	REGION ReadData()
	    //************************************************************************************************ 
	    //从接口读取数据/Read data from interface
	    //************************************************************************************************ 
	    //命令状态/Command Status bits
	    #aRetvalRead[1] := DPRD_DAT(LADDR := "DB_KeyenceCheckerIV3".aDev[#I_nID].Para.nInAdr1, RECORD => #aInput_Byte1);
	    //设备结果/Device Results bits
	    #aRetvalRead[2] := DPRD_DAT(LADDR := "DB_KeyenceCheckerIV3".aDev[#I_nID].Para.nInAdr2, RECORD => #aInput_Byte2);
	    //设备状态/Device status words
	    #aRetvalRead[3] := DPRD_DAT(LADDR := "DB_KeyenceCheckerIV3".aDev[#I_nID].Para.nInAdr3, RECORD => #aInput_Byte3);
	    //设备统计/Device statistics
	    #aRetvalRead[4] := DPRD_DAT(LADDR := "DB_KeyenceCheckerIV3".aDev[#I_nID].Para.nInAdr4, RECORD => #aInput_Byte4);
	    //位置修正结果/Position adjust result
	    #aRetvalRead[5] := DPRD_DAT(LADDR := "DB_KeyenceCheckerIV3".aDev[#I_nID].Para.nInAdr5, RECORD => #aInput_Byte5);
	    //工具1处理结果/Tool1 result
	    #aRetvalRead[6] := DPRD_DAT(LADDR := "DB_KeyenceCheckerIV3".aDev[#I_nID].Para.nInAdr6, RECORD => #aInput_Byte6[0]);
	    //工具2处理结果/Tool2 result
	    #aRetvalRead[7] := DPRD_DAT(LADDR := "DB_KeyenceCheckerIV3".aDev[#I_nID].Para.nInAdr7, RECORD => #aInput_Byte6[1]);
	    //工具3处理结果/Tool3 result
	    #aRetvalRead[8] := DPRD_DAT(LADDR := "DB_KeyenceCheckerIV3".aDev[#I_nID].Para.nInAdr8, RECORD => #aInput_Byte6[2]);
	    //工具4处理结果/Tool4 result
	    #aRetvalRead[9] := DPRD_DAT(LADDR := "DB_KeyenceCheckerIV3".aDev[#I_nID].Para.nInAdr9, RECORD => #aInput_Byte6[3]);
	    //工具5处理结果/Tool5 result
	    #aRetvalRead[10] := DPRD_DAT(LADDR := "DB_KeyenceCheckerIV3".aDev[#I_nID].Para.nInAdr10, RECORD => #aInput_Byte6[4]);
	    //工具6处理结果/Tool6 result
	    #aRetvalRead[11] := DPRD_DAT(LADDR := "DB_KeyenceCheckerIV3".aDev[#I_nID].Para.nInAdr11, RECORD => #aInput_Byte6[5]);
	    //工具7处理结果/Tool7 result
	    #aRetvalRead[12] := DPRD_DAT(LADDR := "DB_KeyenceCheckerIV3".aDev[#I_nID].Para.nInAdr12, RECORD => #aInput_Byte6[6]);
	    //工具8处理结果/Tool8 result
	    #aRetvalRead[13] := DPRD_DAT(LADDR := "DB_KeyenceCheckerIV3".aDev[#I_nID].Para.nInAdr13, RECORD => #aInput_Byte6[7]);
	    //工具9处理结果/Tool9 result
	    #aRetvalRead[14] := DPRD_DAT(LADDR := "DB_KeyenceCheckerIV3".aDev[#I_nID].Para.nInAdr14, RECORD => #aInput_Byte6[8]);
	    //工具10处理结果/Tool10 result
	    #aRetvalRead[15] := DPRD_DAT(LADDR := "DB_KeyenceCheckerIV3".aDev[#I_nID].Para.nInAdr15, RECORD => #aInput_Byte6[9]);
	    //工具11处理结果/Tool11 result
	    #aRetvalRead[16] := DPRD_DAT(LADDR := "DB_KeyenceCheckerIV3".aDev[#I_nID].Para.nInAdr16, RECORD => #aInput_Byte6[10]);
	    //工具12处理结果/Tool12 result
	    #aRetvalRead[17] := DPRD_DAT(LADDR := "DB_KeyenceCheckerIV3".aDev[#I_nID].Para.nInAdr17, RECORD => #aInput_Byte6[11]);
	    //工具13处理结果/Tool13 result
	    #aRetvalRead[18] := DPRD_DAT(LADDR := "DB_KeyenceCheckerIV3".aDev[#I_nID].Para.nInAdr18, RECORD => #aInput_Byte6[12]);
	    //工具14处理结果/Tool14 result
	    #aRetvalRead[19] := DPRD_DAT(LADDR := "DB_KeyenceCheckerIV3".aDev[#I_nID].Para.nInAdr19, RECORD => #aInput_Byte6[13]);
	    //工具15处理结果/Tool15 result
	    #aRetvalRead[20] := DPRD_DAT(LADDR := "DB_KeyenceCheckerIV3".aDev[#I_nID].Para.nInAdr20, RECORD => #aInput_Byte6[14]);
	    //工具16处理结果/Tool16 result
	    #aRetvalRead[21] := DPRD_DAT(LADDR := "DB_KeyenceCheckerIV3".aDev[#I_nID].Para.nInAdr21, RECORD => #aInput_Byte6[15]);
	    //工具17处理结果/Tool1 result
	    #aRetvalRead[6] := DPRD_DAT(LADDR := "DB_KeyenceCheckerIV3".aDev[#I_nID].Para.nInAdr22, RECORD => #aInput_Byte6[16]);
	    //工具18处理结果/Tool2 result
	    #aRetvalRead[7] := DPRD_DAT(LADDR := "DB_KeyenceCheckerIV3".aDev[#I_nID].Para.nInAdr23, RECORD => #aInput_Byte6[17]);
	    //工具19处理结果/Tool3 result
	    #aRetvalRead[8] := DPRD_DAT(LADDR := "DB_KeyenceCheckerIV3".aDev[#I_nID].Para.nInAdr24, RECORD => #aInput_Byte6[18]);
	    //工具20处理结果/Tool4 result
	    #aRetvalRead[9] := DPRD_DAT(LADDR := "DB_KeyenceCheckerIV3".aDev[#I_nID].Para.nInAdr25, RECORD => #aInput_Byte6[19]);
	    //工具21处理结果/Tool5 result
	    #aRetvalRead[10] := DPRD_DAT(LADDR := "DB_KeyenceCheckerIV3".aDev[#I_nID].Para.nInAdr26, RECORD => #aInput_Byte6[20]);
	    //工具22处理结果/Tool6 result
	    #aRetvalRead[11] := DPRD_DAT(LADDR := "DB_KeyenceCheckerIV3".aDev[#I_nID].Para.nInAdr27, RECORD => #aInput_Byte6[21]);
	    //工具23处理结果/Tool7 result
	    #aRetvalRead[12] := DPRD_DAT(LADDR := "DB_KeyenceCheckerIV3".aDev[#I_nID].Para.nInAdr28, RECORD => #aInput_Byte6[22]);
	    //工具24处理结果/Tool8 result
	    #aRetvalRead[13] := DPRD_DAT(LADDR := "DB_KeyenceCheckerIV3".aDev[#I_nID].Para.nInAdr29, RECORD => #aInput_Byte6[23]);
	    //工具25处理结果/Tool9 result
	    #aRetvalRead[14] := DPRD_DAT(LADDR := "DB_KeyenceCheckerIV3".aDev[#I_nID].Para.nInAdr30, RECORD => #aInput_Byte6[24]);
	    //工具26处理结果/Tool10 result
	    #aRetvalRead[15] := DPRD_DAT(LADDR := "DB_KeyenceCheckerIV3".aDev[#I_nID].Para.nInAdr31, RECORD => #aInput_Byte6[25]);
	    //工具27处理结果/Tool11 result
	    #aRetvalRead[16] := DPRD_DAT(LADDR := "DB_KeyenceCheckerIV3".aDev[#I_nID].Para.nInAdr32, RECORD => #aInput_Byte6[26]);
	    //工具28处理结果/Tool12 result
	    #aRetvalRead[17] := DPRD_DAT(LADDR := "DB_KeyenceCheckerIV3".aDev[#I_nID].Para.nInAdr33, RECORD => #aInput_Byte6[27]);
	    //工具29处理结果/Tool13 result
	    #aRetvalRead[18] := DPRD_DAT(LADDR := "DB_KeyenceCheckerIV3".aDev[#I_nID].Para.nInAdr34, RECORD => #aInput_Byte6[28]);
	    //工具30处理结果/Tool14 result
	    #aRetvalRead[19] := DPRD_DAT(LADDR := "DB_KeyenceCheckerIV3".aDev[#I_nID].Para.nInAdr35, RECORD => #aInput_Byte6[29]);
	    //工具31处理结果/Tool15 result
	    #aRetvalRead[20] := DPRD_DAT(LADDR := "DB_KeyenceCheckerIV3".aDev[#I_nID].Para.nInAdr36, RECORD => #aInput_Byte6[30]);
	    //工具32处理结果/Tool16 result
	    #aRetvalRead[21] := DPRD_DAT(LADDR := "DB_KeyenceCheckerIV3".aDev[#I_nID].Para.nInAdr37, RECORD => #aInput_Byte6[31]);
	    //工具33处理结果/Tool1 result
	    #aRetvalRead[6] := DPRD_DAT(LADDR := "DB_KeyenceCheckerIV3".aDev[#I_nID].Para.nInAdr38, RECORD => #aInput_Byte6[32]);
	    //工具34处理结果/Tool2 result
	    #aRetvalRead[7] := DPRD_DAT(LADDR := "DB_KeyenceCheckerIV3".aDev[#I_nID].Para.nInAdr39, RECORD => #aInput_Byte6[33]);
	    //工具35处理结果/Tool3 result
	    #aRetvalRead[8] := DPRD_DAT(LADDR := "DB_KeyenceCheckerIV3".aDev[#I_nID].Para.nInAdr40, RECORD => #aInput_Byte6[34]);
	    //工具36处理结果/Tool4 result
	    #aRetvalRead[9] := DPRD_DAT(LADDR := "DB_KeyenceCheckerIV3".aDev[#I_nID].Para.nInAdr41, RECORD => #aInput_Byte6[35]);
	    //工具37处理结果/Tool5 result
	    #aRetvalRead[10] := DPRD_DAT(LADDR := "DB_KeyenceCheckerIV3".aDev[#I_nID].Para.nInAdr42, RECORD => #aInput_Byte6[36]);
	    //工具38处理结果/Tool6 result
	    #aRetvalRead[11] := DPRD_DAT(LADDR := "DB_KeyenceCheckerIV3".aDev[#I_nID].Para.nInAdr43, RECORD => #aInput_Byte6[37]);
	    //工具39处理结果/Tool7 result
	    #aRetvalRead[12] := DPRD_DAT(LADDR := "DB_KeyenceCheckerIV3".aDev[#I_nID].Para.nInAdr44, RECORD => #aInput_Byte6[38]);
	    //工具40处理结果/Tool8 result
	    #aRetvalRead[13] := DPRD_DAT(LADDR := "DB_KeyenceCheckerIV3".aDev[#I_nID].Para.nInAdr45, RECORD => #aInput_Byte6[39]);
	    //工具41处理结果/Tool9 result
	    #aRetvalRead[14] := DPRD_DAT(LADDR := "DB_KeyenceCheckerIV3".aDev[#I_nID].Para.nInAdr46, RECORD => #aInput_Byte6[40]);
	    //工具42处理结果/Tool10 result
	    #aRetvalRead[15] := DPRD_DAT(LADDR := "DB_KeyenceCheckerIV3".aDev[#I_nID].Para.nInAdr47, RECORD => #aInput_Byte6[41]);
	    //工具43处理结果/Tool11 result
	    #aRetvalRead[16] := DPRD_DAT(LADDR := "DB_KeyenceCheckerIV3".aDev[#I_nID].Para.nInAdr48, RECORD => #aInput_Byte6[42]);
	    //工具44处理结果/Tool12 result
	    #aRetvalRead[17] := DPRD_DAT(LADDR := "DB_KeyenceCheckerIV3".aDev[#I_nID].Para.nInAdr49, RECORD => #aInput_Byte6[43]);
	    //工具45处理结果/Tool13 result
	    #aRetvalRead[18] := DPRD_DAT(LADDR := "DB_KeyenceCheckerIV3".aDev[#I_nID].Para.nInAdr50, RECORD => #aInput_Byte6[44]);
	    //工具46处理结果/Tool14 result
	    #aRetvalRead[19] := DPRD_DAT(LADDR := "DB_KeyenceCheckerIV3".aDev[#I_nID].Para.nInAdr51, RECORD => #aInput_Byte6[45]);
	    //工具47处理结果/Tool15 result
	    #aRetvalRead[20] := DPRD_DAT(LADDR := "DB_KeyenceCheckerIV3".aDev[#I_nID].Para.nInAdr52, RECORD => #aInput_Byte6[46]);
	    //工具48处理结果/Tool16 result
	    #aRetvalRead[21] := DPRD_DAT(LADDR := "DB_KeyenceCheckerIV3".aDev[#I_nID].Para.nInAdr53, RECORD => #aInput_Byte6[47]);
	    //工具49处理结果/Tool1 result
	    #aRetvalRead[6] := DPRD_DAT(LADDR := "DB_KeyenceCheckerIV3".aDev[#I_nID].Para.nInAdr54, RECORD => #aInput_Byte6[48]);
	    //工具50处理结果/Tool2 result
	    #aRetvalRead[7] := DPRD_DAT(LADDR := "DB_KeyenceCheckerIV3".aDev[#I_nID].Para.nInAdr55, RECORD => #aInput_Byte6[49]);
	    //工具51处理结果/Tool3 result
	    #aRetvalRead[8] := DPRD_DAT(LADDR := "DB_KeyenceCheckerIV3".aDev[#I_nID].Para.nInAdr56, RECORD => #aInput_Byte6[50]);
	    //工具52处理结果/Tool4 result
	    #aRetvalRead[9] := DPRD_DAT(LADDR := "DB_KeyenceCheckerIV3".aDev[#I_nID].Para.nInAdr57, RECORD => #aInput_Byte6[51]);
	    //工具53处理结果/Tool5 result
	    #aRetvalRead[10] := DPRD_DAT(LADDR := "DB_KeyenceCheckerIV3".aDev[#I_nID].Para.nInAdr58, RECORD => #aInput_Byte6[52]);
	    //工具54处理结果/Tool6 result
	    #aRetvalRead[11] := DPRD_DAT(LADDR := "DB_KeyenceCheckerIV3".aDev[#I_nID].Para.nInAdr59, RECORD => #aInput_Byte6[53]);
	    //工具55处理结果/Tool7 result
	    #aRetvalRead[12] := DPRD_DAT(LADDR := "DB_KeyenceCheckerIV3".aDev[#I_nID].Para.nInAdr60, RECORD => #aInput_Byte6[54]);
	    //工具56处理结果/Tool8 result
	    #aRetvalRead[13] := DPRD_DAT(LADDR := "DB_KeyenceCheckerIV3".aDev[#I_nID].Para.nInAdr61, RECORD => #aInput_Byte6[55]);
	    //工具57处理结果/Tool9 result
	    #aRetvalRead[14] := DPRD_DAT(LADDR := "DB_KeyenceCheckerIV3".aDev[#I_nID].Para.nInAdr62, RECORD => #aInput_Byte6[56]);
	    //工具58处理结果/Tool10 result
	    #aRetvalRead[15] := DPRD_DAT(LADDR := "DB_KeyenceCheckerIV3".aDev[#I_nID].Para.nInAdr63, RECORD => #aInput_Byte6[57]);
	    //工具59处理结果/Tool11 result
	    #aRetvalRead[16] := DPRD_DAT(LADDR := "DB_KeyenceCheckerIV3".aDev[#I_nID].Para.nInAdr64, RECORD => #aInput_Byte6[58]);
	    //工具60处理结果/Tool12 result
	    #aRetvalRead[17] := DPRD_DAT(LADDR := "DB_KeyenceCheckerIV3".aDev[#I_nID].Para.nInAdr65, RECORD => #aInput_Byte6[59]);
	    //工具61处理结果/Tool13 result
	    #aRetvalRead[18] := DPRD_DAT(LADDR := "DB_KeyenceCheckerIV3".aDev[#I_nID].Para.nInAdr66, RECORD => #aInput_Byte6[60]);
	    //工具62处理结果/Tool14 result
	    #aRetvalRead[19] := DPRD_DAT(LADDR := "DB_KeyenceCheckerIV3".aDev[#I_nID].Para.nInAdr67, RECORD => #aInput_Byte6[61]);
	    //工具63处理结果/Tool15 result
	    #aRetvalRead[20] := DPRD_DAT(LADDR := "DB_KeyenceCheckerIV3".aDev[#I_nID].Para.nInAdr68, RECORD => #aInput_Byte6[62]);
	    //工具64处理结果/Tool16 result
	    #aRetvalRead[21] := DPRD_DAT(LADDR := "DB_KeyenceCheckerIV3".aDev[#I_nID].Para.nInAdr69, RECORD => #aInput_Byte6[63]);
	    //设备结果/Device Results bits
	    #aRetvalRead[22] := DPRD_DAT(LADDR := "DB_KeyenceCheckerIV3".aDev[#I_nID].Para.nInAdr70, RECORD => #aInput_Byte7);
	    "DB_KeyenceCheckerIV3".aDev[#I_nID].Common.nID := #I_nID;
	END_REGION
	
	REGION CopyReadData()
	    ///************************************************************************************************
	    //分配输入数据/Asignment of the intput data (Statusword)
	    //************************************************************************************************
	    //命令状态/Command status bits
	    //Address 0
	    #nByte := #aInput_Byte1[0];
	    "DB_KeyenceCheckerIV3".aDev[#I_nID].In.CommandStatus.bTriggerResponse := #nByte.%X0;
	    "DB_KeyenceCheckerIV3".aDev[#I_nID].In.CommandStatus.bMasterImageRegistration := #nByte.%X1;
	    "DB_KeyenceCheckerIV3".aDev[#I_nID].In.CommandStatus.bProgramSwitchingResponse := #nByte.%X2;
	    "DB_KeyenceCheckerIV3".aDev[#I_nID].In.CommandStatus.bWarningClearResponse := #nByte.%X3;
	    "DB_KeyenceCheckerIV3".aDev[#I_nID].In.CommandStatus.bStatisticsResetResponse := #nByte.%X4;
	    "DB_KeyenceCheckerIV3".aDev[#I_nID].In.CommandStatus.bBufferClearResponse := #nByte.%X5;
	    "DB_KeyenceCheckerIV3".aDev[#I_nID].In.CommandStatus.bSDCardStopSaveResponse := #nByte.%X6;
	    "DB_KeyenceCheckerIV3".aDev[#I_nID].In.CommandStatus.bChangeParameterResponse := #nByte.%X7;
	    //Address 1
	    #nByte := #aInput_Byte1[1];
	    "DB_KeyenceCheckerIV3".aDev[#I_nID].In.CommandStatus.bTriggerFailed := #nByte.%X0;
	    "DB_KeyenceCheckerIV3".aDev[#I_nID].In.CommandStatus.bMasterImageRegistrationFailed := #nByte.%X1;
	    "DB_KeyenceCheckerIV3".aDev[#I_nID].In.CommandStatus.bProgramSwitchingFailed := #nByte.%X2;
	    "DB_KeyenceCheckerIV3".aDev[#I_nID].In.CommandStatus.bReserved1 := #nByte.%X3;
	    "DB_KeyenceCheckerIV3".aDev[#I_nID].In.CommandStatus.bReserved2 := #nByte.%X4;
	    "DB_KeyenceCheckerIV3".aDev[#I_nID].In.CommandStatus.bReserved3 := #nByte.%X5;
	    "DB_KeyenceCheckerIV3".aDev[#I_nID].In.CommandStatus.bSDCardStopSaveFailed := #nByte.%X6;
	    "DB_KeyenceCheckerIV3".aDev[#I_nID].In.CommandStatus.bChangeParameterFailed := #nByte.%X7;
	    //Address 2 
	    #nByte := #aInput_Byte1[2];
	    "DB_KeyenceCheckerIV3".aDev[#I_nID].In.CommandStatus.bResultAvailable := #nByte.%X0;
	    "DB_KeyenceCheckerIV3".aDev[#I_nID].In.CommandStatus.bResultUpdateComplete := #nByte.%X1;
	    "DB_KeyenceCheckerIV3".aDev[#I_nID].In.CommandStatus.bBusy := #nByte.%X2;
	    "DB_KeyenceCheckerIV3".aDev[#I_nID].In.CommandStatus.bImaging := #nByte.%X3;
	    "DB_KeyenceCheckerIV3".aDev[#I_nID].In.CommandStatus.bRun := #nByte.%X4;
	    "DB_KeyenceCheckerIV3".aDev[#I_nID].In.CommandStatus.bReady := #nByte.%X5;
	    "DB_KeyenceCheckerIV3".aDev[#I_nID].In.CommandStatus.bReserved4 := #nByte.%X6;
	    "DB_KeyenceCheckerIV3".aDev[#I_nID].In.CommandStatus.bSDCardStatus := #nByte.%X7;
	    //Address 3
	    #nByte := #aInput_Byte1[3];
	    "DB_KeyenceCheckerIV3".aDev[#I_nID].In.CommandStatus.bClassificationModeInformation := #nByte.%X0;
	    "DB_KeyenceCheckerIV3".aDev[#I_nID].In.CommandStatus.bReserved5 := #nByte.%X1;
	    "DB_KeyenceCheckerIV3".aDev[#I_nID].In.CommandStatus.bReserved6 := #nByte.%X2;
	    "DB_KeyenceCheckerIV3".aDev[#I_nID].In.CommandStatus.bReserved7 := #nByte.%X3;
	    "DB_KeyenceCheckerIV3".aDev[#I_nID].In.CommandStatus.bSDCardStorageShortage := #nByte.%X4;
	    "DB_KeyenceCheckerIV3".aDev[#I_nID].In.CommandStatus.bBufferOverrun := #nByte.%X5;
	    "DB_KeyenceCheckerIV3".aDev[#I_nID].In.CommandStatus.bWarning := #nByte.%X6;
	    "DB_KeyenceCheckerIV3".aDev[#I_nID].In.CommandStatus.bError := #nByte.%X7;
	    
	    //设备结果/Device Results Bits
	    //Address 0
	    #nByte := #aInput_Byte2[0];
	    "DB_KeyenceCheckerIV3".aDev[#I_nID].In.DeviceResults.bOverallJudgmentOK := #nByte.%X0;
	    "DB_KeyenceCheckerIV3".aDev[#I_nID].In.DeviceResults.bPositionCorrection := #nByte.%X1;
	    "DB_KeyenceCheckerIV3".aDev[#I_nID].In.DeviceResults.bLogic1 := #nByte.%X2;
	    "DB_KeyenceCheckerIV3".aDev[#I_nID].In.DeviceResults.bLogic2 := #nByte.%X3;
	    "DB_KeyenceCheckerIV3".aDev[#I_nID].In.DeviceResults.bLogic3 := #nByte.%X4;
	    "DB_KeyenceCheckerIV3".aDev[#I_nID].In.DeviceResults.bLogic4 := #nByte.%X5;
	    "DB_KeyenceCheckerIV3".aDev[#I_nID].In.DeviceResults.bOverallJudgmentNG := #nByte.%X6;
	    "DB_KeyenceCheckerIV3".aDev[#I_nID].In.DeviceResults.bReserved1 := #nByte.%X7;
	    //Address 1
	    #nByte := #aInput_Byte2[1];
	    "DB_KeyenceCheckerIV3".aDev[#I_nID].In.DeviceResults.nReserved2 := #nByte;
	    //Address 2
	    #nByte := #aInput_Byte2[2];
	    "DB_KeyenceCheckerIV3".aDev[#I_nID].In.DeviceResults.aToolResult[1] := #nByte.%X0;
	    "DB_KeyenceCheckerIV3".aDev[#I_nID].In.DeviceResults.aToolResult[2] := #nByte.%X1;
	    "DB_KeyenceCheckerIV3".aDev[#I_nID].In.DeviceResults.aToolResult[3] := #nByte.%X2;
	    "DB_KeyenceCheckerIV3".aDev[#I_nID].In.DeviceResults.aToolResult[4] := #nByte.%X3;
	    "DB_KeyenceCheckerIV3".aDev[#I_nID].In.DeviceResults.aToolResult[5] := #nByte.%X4;
	    "DB_KeyenceCheckerIV3".aDev[#I_nID].In.DeviceResults.aToolResult[6] := #nByte.%X5;
	    "DB_KeyenceCheckerIV3".aDev[#I_nID].In.DeviceResults.aToolResult[7] := #nByte.%X6;
	    "DB_KeyenceCheckerIV3".aDev[#I_nID].In.DeviceResults.aToolResult[8] := #nByte.%X7;
	    //Address 3
	    #nByte := #aInput_Byte2[3];
	    "DB_KeyenceCheckerIV3".aDev[#I_nID].In.DeviceResults.aToolResult[9] := #nByte.%X0;
	    "DB_KeyenceCheckerIV3".aDev[#I_nID].In.DeviceResults.aToolResult[10] := #nByte.%X1;
	    "DB_KeyenceCheckerIV3".aDev[#I_nID].In.DeviceResults.aToolResult[11] := #nByte.%X2;
	    "DB_KeyenceCheckerIV3".aDev[#I_nID].In.DeviceResults.aToolResult[12] := #nByte.%X3;
	    "DB_KeyenceCheckerIV3".aDev[#I_nID].In.DeviceResults.aToolResult[13] := #nByte.%X4;
	    "DB_KeyenceCheckerIV3".aDev[#I_nID].In.DeviceResults.aToolResult[14] := #nByte.%X5;
	    "DB_KeyenceCheckerIV3".aDev[#I_nID].In.DeviceResults.aToolResult[15] := #nByte.%X6;
	    "DB_KeyenceCheckerIV3".aDev[#I_nID].In.DeviceResults.aToolResult[16] := #nByte.%X7;
	    
	    //设备状态/Device status words
	    //错误编号/Error number
	    #aWord[0] := #aInput_Byte3[0];
	    #aWord[1] := #aInput_Byte3[1];
	    "DB_KeyenceCheckerIV3".aDev[#I_nID].In."DeviceStatus".nErrorNo := #nWord;
	    //警报编号/Warning number
	    #aWord[0] := #aInput_Byte3[2];
	    #aWord[1] := #aInput_Byte3[3];
	    "DB_KeyenceCheckerIV3".aDev[#I_nID].In."DeviceStatus".nWarningNo := #nWord;
	    //剩余缓存数/Number of remaining buffers
	    #aWord[0] := #aInput_Byte3[4];
	    #aWord[1] := #aInput_Byte3[5];
	    "DB_KeyenceCheckerIV3".aDev[#I_nID].In."DeviceStatus".nNumberOfRemainingBuffers := #nWord;
	    //设定校验和/Check sum
	    #aWord[0] := #aInput_Byte3[6];
	    #aWord[1] := #aInput_Byte3[7];
	    "DB_KeyenceCheckerIV3".aDev[#I_nID].In."DeviceStatus".nChecksum := #nWord;
	    //当前程序编号/Current program number
	    #aWord[0] := #aInput_Byte3[8];
	    #aWord[1] := #aInput_Byte3[9];
	    "DB_KeyenceCheckerIV3".aDev[#I_nID].In."DeviceStatus".nCurrentProgramNo := #nWord;
	    //判断时程序编号/Program number during judgment
	    #aWord[0] := #aInput_Byte3[10];
	    #aWord[1] := #aInput_Byte3[11];
	    "DB_KeyenceCheckerIV3".aDev[#I_nID].In."DeviceStatus".nProgramNoDuringJudgment := #nWord;
	    //结果编号/Result number
	    #aWord[0] := #aInput_Byte3[12];
	    #aWord[1] := #aInput_Byte3[13];
	    "DB_KeyenceCheckerIV3".aDev[#I_nID].In."DeviceStatus".nResultNo := #nWord;
	    //处理时间/Processing time
	    #aWord[0] := #aInput_Byte3[14];
	    #aWord[1] := #aInput_Byte3[15];
	    "DB_KeyenceCheckerIV3".aDev[#I_nID].In."DeviceStatus".nProcessingtime := #nWord;
	    
	    //设备统计/Device Statistics
	    //最大处理时间/Processing time max
	    #aWord[0] := #aInput_Byte4[0];
	    #aWord[1] := #aInput_Byte4[1];
	    "DB_KeyenceCheckerIV3".aDev[#I_nID].In."DeviceStatistics".nProcessingTimeMAX := #nWord;
	    //最小处理时间/Processing time min
	    #aWord[0] := #aInput_Byte4[2];
	    #aWord[1] := #aInput_Byte4[3];
	    "DB_KeyenceCheckerIV3".aDev[#I_nID].In."DeviceStatistics".nProcessingTimeMIN := #nWord;
	    //平均处理时间/Processing time average
	    #aWord[0] := #aInput_Byte4[4];
	    #aWord[1] := #aInput_Byte4[5];
	    "DB_KeyenceCheckerIV3".aDev[#I_nID].In."DeviceStatistics".nProcessingTimeAVE := #nWord;
	    //系统预约/Reserved by system
	    #aWord[0] := #aInput_Byte4[6];
	    #aWord[1] := #aInput_Byte4[7];
	    "DB_KeyenceCheckerIV3".aDev[#I_nID].In."DeviceStatistics".nReserved1 := #nWord;
	    //触发次数/Number of triggers
	    #aDWord[0] := #aInput_Byte4[8];
	    #aDWord[1] := #aInput_Byte4[9];
	    #aDWord[2] := #aInput_Byte4[10];
	    #aDWord[3] := #aInput_Byte4[11];
	    "DB_KeyenceCheckerIV3".aDev[#I_nID].In."DeviceStatistics".nNumberOfTriggers := #nDWord;
	    //OK 次数或分类次数/Number of OKs OR Classification number
	    #aDWord[0] := #aInput_Byte4[12];
	    #aDWord[1] := #aInput_Byte4[13];
	    #aDWord[2] := #aInput_Byte4[14];
	    #aDWord[3] := #aInput_Byte4[15];
	    "DB_KeyenceCheckerIV3".aDev[#I_nID].In."DeviceStatistics".nNumberOfOKs := #nDWord;
	    //NG 次数/Number of NGs
	    #aDWord[0] := #aInput_Byte4[16];
	    #aDWord[1] := #aInput_Byte4[17];
	    #aDWord[2] := #aInput_Byte4[18];
	    #aDWord[3] := #aInput_Byte4[19];
	    "DB_KeyenceCheckerIV3".aDev[#I_nID].In."DeviceStatistics".nNumberOfNGs := #nDWord;
	    //触发错误次数/Number of trigger errors
	    #aDWord[0] := #aInput_Byte4[20];
	    #aDWord[1] := #aInput_Byte4[21];
	    #aDWord[2] := #aInput_Byte4[22];
	    #aDWord[3] := #aInput_Byte4[23];
	    "DB_KeyenceCheckerIV3".aDev[#I_nID].In."DeviceStatistics".nNumberOfTriggerErrors := #nDWord;
	    //系统预约/Reserved by system
	    #aDWord[0] := #aInput_Byte4[24];
	    #aDWord[1] := #aInput_Byte4[25];
	    #aDWord[2] := #aInput_Byte4[26];
	    #aDWord[3] := #aInput_Byte4[27];
	    "DB_KeyenceCheckerIV3".aDev[#I_nID].In."DeviceStatistics".nReserved2 := #nDWord;
	    
	    //位置修正结果/Position Adjust Result
	    //位置修正分数/Position correction tool matching rate
	    #aWord[0] := #aInput_Byte5[0];
	    #aWord[1] := #aInput_Byte5[1];
	    "DB_KeyenceCheckerIV3".aDev[#I_nID].In."PositionAdjustResult".nPositionCorrectionToolMatchingRate := #nWord;
	    //最大位置修正分数/Position correction tool matching rate max
	    #aWord[0] := #aInput_Byte5[2];
	    #aWord[1] := #aInput_Byte5[3];
	    "DB_KeyenceCheckerIV3".aDev[#I_nID].In."PositionAdjustResult".nPositionCorrectionToolMatchingRateMAX := #nWord;
	    //最小位置修正分数/Position correction tool matching rate min
	    #aWord[0] := #aInput_Byte5[4];
	    #aWord[1] := #aInput_Byte5[5];
	    "DB_KeyenceCheckerIV3".aDev[#I_nID].In."PositionAdjustResult".nPositionCorrectionToolMatchingRateMIN := #nWord;
	    //位置修正分数下限阈值/Position correction tool threshold
	    #aWord[0] := #aInput_Byte5[6];
	    #aWord[1] := #aInput_Byte5[7];
	    "DB_KeyenceCheckerIV3".aDev[#I_nID].In."PositionAdjustResult".nPositionCorrectionToolThreshold := #nWord;
	    //系统预约/Reserved by system
	    #aWord[0] := #aInput_Byte5[8];
	    #aWord[1] := #aInput_Byte5[9];
	    "DB_KeyenceCheckerIV3".aDev[#I_nID].In."PositionAdjustResult".nReserved1 := #nWord;
	    //系统预约/Reserved by system
	    #aWord[0] := #aInput_Byte5[10];
	    #aWord[1] := #aInput_Byte5[11];
	    "DB_KeyenceCheckerIV3".aDev[#I_nID].In."PositionAdjustResult".nReserved2 := #nWord;
	    //系统预约/Reserved by system
	    #aWord[0] := #aInput_Byte5[12];
	    #aWord[1] := #aInput_Byte5[13];
	    "DB_KeyenceCheckerIV3".aDev[#I_nID].In."PositionAdjustResult".nReserved3 := #nWord;
	    //系统预约/Reserved by system
	    #aWord[0] := #aInput_Byte5[14];
	    #aWord[1] := #aInput_Byte5[15];
	    "DB_KeyenceCheckerIV3".aDev[#I_nID].In."PositionAdjustResult".nReserved4 := #nWord;
	    //系统预约/Reserved by system
	    #aWord[0] := #aInput_Byte5[16];
	    #aWord[1] := #aInput_Byte5[17];
	    "DB_KeyenceCheckerIV3".aDev[#I_nID].In."PositionAdjustResult".nReserved5 := #nWord;
	    //系统预约/Reserved by system
	    #aWord[0] := #aInput_Byte5[18];
	    #aWord[1] := #aInput_Byte5[19];
	    "DB_KeyenceCheckerIV3".aDev[#I_nID].In."PositionAdjustResult".nReserved6 := #nWord;
	    
	    //工具处理结果/Tool Results
	    FOR #nIdx := 1 TO 64 BY 1 DO
	        //工具相似度/Tool matching rate
	        #aWord[0] := #aInput_Byte6[#nIdx - 1].bInput_Byte0;
	        #aWord[1] := #aInput_Byte6[#nIdx - 1].bInput_Byte1;
	        "DB_KeyenceCheckerIV3".aDev[#I_nID].In.ToolResult[#nIdx].nToolMatchingRate := #nWord;
	        //最大工具相似度/Tool matching rate max
	        #aWord[0] := #aInput_Byte6[#nIdx - 1].bInput_Byte2;
	        #aWord[1] := #aInput_Byte6[#nIdx - 1].bInput_Byte3;
	        "DB_KeyenceCheckerIV3".aDev[#I_nID].In.ToolResult[#nIdx].nToolMatchingRateMAX := #nWord;
	        //最小工具相似度/Tool matching rate min
	        #aWord[0] := #aInput_Byte6[#nIdx - 1].bInput_Byte4;
	        #aWord[1] := #aInput_Byte6[#nIdx - 1].bInput_Byte5;
	        "DB_KeyenceCheckerIV3".aDev[#I_nID].In.ToolResult[#nIdx].nToolMatchingRateMIN := #nWord;
	        //工具下限阈值/Tool lower limit value
	        #aWord[0] := #aInput_Byte6[#nIdx - 1].bInput_Byte6;
	        #aWord[1] := #aInput_Byte6[#nIdx - 1].bInput_Byte7;
	        "DB_KeyenceCheckerIV3".aDev[#I_nID].In.ToolResult[#nIdx].nToolLowerLimitValue := #nWord;
	        //工具上限阈值/Tool upper limit value
	        #aWord[0] := #aInput_Byte6[#nIdx - 1].bInput_Byte8;
	        #aWord[1] := #aInput_Byte6[#nIdx - 1].bInput_Byte9;
	        "DB_KeyenceCheckerIV3".aDev[#I_nID].In.ToolResult[#nIdx].nToolUpperLimitValue := #nWord;
	        //小数点位置/Decimal position
	        #aWord[0] := #aInput_Byte6[#nIdx - 1].bInput_Byte10;
	        #aWord[1] := #aInput_Byte6[#nIdx - 1].bInput_Byte11;
	        "DB_KeyenceCheckerIV3".aDev[#I_nID].In.ToolResult[#nIdx].nDecimalPosition := #nWord;
	        //间距当前值 MAX&彩色识别 H（色相）/Pitch present value MAX&color average H (hue)
	        #aWord[0] := #aInput_Byte6[#nIdx - 1].bInput_Byte12;
	        #aWord[1] := #aInput_Byte6[#nIdx - 1].bInput_Byte13;
	        "DB_KeyenceCheckerIV3".aDev[#I_nID].In.ToolResult[#nIdx]."nPitchPresentValueMAX/ColorAverageH (hue)" := #nWord;
	        //间距当前值 MIN&彩色识别 S（彩度）/Pitch present value MIN&color average S
	        #aWord[0] := #aInput_Byte6[#nIdx - 1].bInput_Byte14;
	        #aWord[1] := #aInput_Byte6[#nIdx - 1].bInput_Byte15;
	        "DB_KeyenceCheckerIV3".aDev[#I_nID].In.ToolResult[#nIdx]."nPitchPresentValueMIN/ColorAverageS(saturation)" := #nWord;
	        //间距数量&彩色识别 V（彩度）&亮度平均亮度/Number of pitches&color average V (brightness)&brightness average 
	        #aWord[0] := #aInput_Byte6[#nIdx - 1].bInput_Byte16;
	        #aWord[1] := #aInput_Byte6[#nIdx - 1].bInput_Byte17;
	        "DB_KeyenceCheckerIV3".aDev[#I_nID].In.ToolResult[#nIdx]."nNumberOfPitches/ColorAverageV(brightness)/BrightnessAverage" := #nWord;
	        //系统预约/Reserved by system
	        #aWord[0] := #aInput_Byte6[#nIdx - 1].bInput_Byte18;
	        #aWord[1] := #aInput_Byte6[#nIdx - 1].bInput_Byte19;
	        "DB_KeyenceCheckerIV3".aDev[#I_nID].In.ToolResult[#nIdx].nReserved1 := #nWord;
	    END_FOR;
	    
	    //设备结果/Device Results Bits 
	    //主控编号/The master number
	    #aWord[0] := #aInput_Byte7[0];
	    #aWord[1] := #aInput_Byte7[1];
	    "DB_KeyenceCheckerIV3".aDev[#I_nID].In.ExtendedDeviceResult.nMasterNumber := #nWord;
	    //Address 1
	    #nByte := #aInput_Byte7[2];
	    "DB_KeyenceCheckerIV3".aDev[#I_nID].In.ExtendedDeviceResult.aToolResult[17] := #nByte.%X0;
	    "DB_KeyenceCheckerIV3".aDev[#I_nID].In.ExtendedDeviceResult.aToolResult[18] := #nByte.%X1;
	    "DB_KeyenceCheckerIV3".aDev[#I_nID].In.ExtendedDeviceResult.aToolResult[19] := #nByte.%X2;
	    "DB_KeyenceCheckerIV3".aDev[#I_nID].In.ExtendedDeviceResult.aToolResult[20] := #nByte.%X3;
	    "DB_KeyenceCheckerIV3".aDev[#I_nID].In.ExtendedDeviceResult.aToolResult[21] := #nByte.%X4;
	    "DB_KeyenceCheckerIV3".aDev[#I_nID].In.ExtendedDeviceResult.aToolResult[22] := #nByte.%X5;
	    "DB_KeyenceCheckerIV3".aDev[#I_nID].In.ExtendedDeviceResult.aToolResult[23] := #nByte.%X6;
	    "DB_KeyenceCheckerIV3".aDev[#I_nID].In.ExtendedDeviceResult.aToolResult[24] := #nByte.%X7;
	    //Address 2
	    #nByte := #aInput_Byte7[3];
	    "DB_KeyenceCheckerIV3".aDev[#I_nID].In.ExtendedDeviceResult.aToolResult[25] := #nByte.%X0;
	    "DB_KeyenceCheckerIV3".aDev[#I_nID].In.ExtendedDeviceResult.aToolResult[26] := #nByte.%X1;
	    "DB_KeyenceCheckerIV3".aDev[#I_nID].In.ExtendedDeviceResult.aToolResult[27] := #nByte.%X2;
	    "DB_KeyenceCheckerIV3".aDev[#I_nID].In.ExtendedDeviceResult.aToolResult[28] := #nByte.%X3;
	    "DB_KeyenceCheckerIV3".aDev[#I_nID].In.ExtendedDeviceResult.aToolResult[29] := #nByte.%X4;
	    "DB_KeyenceCheckerIV3".aDev[#I_nID].In.ExtendedDeviceResult.aToolResult[30] := #nByte.%X5;
	    "DB_KeyenceCheckerIV3".aDev[#I_nID].In.ExtendedDeviceResult.aToolResult[31] := #nByte.%X6;
	    "DB_KeyenceCheckerIV3".aDev[#I_nID].In.ExtendedDeviceResult.aToolResult[32] := #nByte.%X7;
	    //Address 3
	    #nByte := #aInput_Byte7[4];
	    "DB_KeyenceCheckerIV3".aDev[#I_nID].In.ExtendedDeviceResult.aToolResult[33] := #nByte.%X0;
	    "DB_KeyenceCheckerIV3".aDev[#I_nID].In.ExtendedDeviceResult.aToolResult[34] := #nByte.%X1;
	    "DB_KeyenceCheckerIV3".aDev[#I_nID].In.ExtendedDeviceResult.aToolResult[35] := #nByte.%X2;
	    "DB_KeyenceCheckerIV3".aDev[#I_nID].In.ExtendedDeviceResult.aToolResult[36] := #nByte.%X3;
	    "DB_KeyenceCheckerIV3".aDev[#I_nID].In.ExtendedDeviceResult.aToolResult[37] := #nByte.%X4;
	    "DB_KeyenceCheckerIV3".aDev[#I_nID].In.ExtendedDeviceResult.aToolResult[38] := #nByte.%X5;
	    "DB_KeyenceCheckerIV3".aDev[#I_nID].In.ExtendedDeviceResult.aToolResult[39] := #nByte.%X6;
	    "DB_KeyenceCheckerIV3".aDev[#I_nID].In.ExtendedDeviceResult.aToolResult[40] := #nByte.%X7;
	    //Address 4
	    #nByte := #aInput_Byte7[5];
	    "DB_KeyenceCheckerIV3".aDev[#I_nID].In.ExtendedDeviceResult.aToolResult[41] := #nByte.%X0;
	    "DB_KeyenceCheckerIV3".aDev[#I_nID].In.ExtendedDeviceResult.aToolResult[42] := #nByte.%X1;
	    "DB_KeyenceCheckerIV3".aDev[#I_nID].In.ExtendedDeviceResult.aToolResult[43] := #nByte.%X2;
	    "DB_KeyenceCheckerIV3".aDev[#I_nID].In.ExtendedDeviceResult.aToolResult[44] := #nByte.%X3;
	    "DB_KeyenceCheckerIV3".aDev[#I_nID].In.ExtendedDeviceResult.aToolResult[45] := #nByte.%X4;
	    "DB_KeyenceCheckerIV3".aDev[#I_nID].In.ExtendedDeviceResult.aToolResult[46] := #nByte.%X5;
	    "DB_KeyenceCheckerIV3".aDev[#I_nID].In.ExtendedDeviceResult.aToolResult[47] := #nByte.%X6;
	    "DB_KeyenceCheckerIV3".aDev[#I_nID].In.ExtendedDeviceResult.aToolResult[48] := #nByte.%X7;
	    //Address 5
	    #nByte := #aInput_Byte7[6];
	    "DB_KeyenceCheckerIV3".aDev[#I_nID].In.ExtendedDeviceResult.aToolResult[49] := #nByte.%X0;
	    "DB_KeyenceCheckerIV3".aDev[#I_nID].In.ExtendedDeviceResult.aToolResult[50] := #nByte.%X1;
	    "DB_KeyenceCheckerIV3".aDev[#I_nID].In.ExtendedDeviceResult.aToolResult[51] := #nByte.%X2;
	    "DB_KeyenceCheckerIV3".aDev[#I_nID].In.ExtendedDeviceResult.aToolResult[52] := #nByte.%X3;
	    "DB_KeyenceCheckerIV3".aDev[#I_nID].In.ExtendedDeviceResult.aToolResult[53] := #nByte.%X4;
	    "DB_KeyenceCheckerIV3".aDev[#I_nID].In.ExtendedDeviceResult.aToolResult[54] := #nByte.%X5;
	    "DB_KeyenceCheckerIV3".aDev[#I_nID].In.ExtendedDeviceResult.aToolResult[55] := #nByte.%X6;
	    "DB_KeyenceCheckerIV3".aDev[#I_nID].In.ExtendedDeviceResult.aToolResult[56] := #nByte.%X7;
	    //Address 6
	    #nByte := #aInput_Byte7[7];
	    "DB_KeyenceCheckerIV3".aDev[#I_nID].In.ExtendedDeviceResult.aToolResult[57] := #nByte.%X0;
	    "DB_KeyenceCheckerIV3".aDev[#I_nID].In.ExtendedDeviceResult.aToolResult[58] := #nByte.%X1;
	    "DB_KeyenceCheckerIV3".aDev[#I_nID].In.ExtendedDeviceResult.aToolResult[59] := #nByte.%X2;
	    "DB_KeyenceCheckerIV3".aDev[#I_nID].In.ExtendedDeviceResult.aToolResult[60] := #nByte.%X3;
	    "DB_KeyenceCheckerIV3".aDev[#I_nID].In.ExtendedDeviceResult.aToolResult[61] := #nByte.%X4;
	    "DB_KeyenceCheckerIV3".aDev[#I_nID].In.ExtendedDeviceResult.aToolResult[62] := #nByte.%X5;
	    "DB_KeyenceCheckerIV3".aDev[#I_nID].In.ExtendedDeviceResult.aToolResult[63] := #nByte.%X6;
	    "DB_KeyenceCheckerIV3".aDev[#I_nID].In.ExtendedDeviceResult.aToolResult[64] := #nByte.%X7;
	END_REGION
	
	REGION CallAdditionalFunctionBlock()
	    //************************************************************************************************
	    //调用外部功能块/Call additional function block
	    //************************************************************************************************
	END_REGION
	
	REGION ErrorMessages()
	    //************************************************************************************************
	    //错误信息/Error messages
	    //************************************************************************************************
	    //复位错误信息/Reset error messages
	    IF "DB_KeyenceCheckerIV3".aDev[#I_nID].Common.bReset AND
	        "DB_KeyenceCheckerIV3".aDev[#I_nID].Common.bError
	    THEN
	        "DB_KeyenceCheckerIV3".aDev[#I_nID].Common.nErrorNo := 0;
	        "DB_KeyenceCheckerIV3".aDev[#I_nID].Common.bError := FALSE;
	        "DB_KeyenceCheckerIV3".aDev[#I_nID].Out.CommandControl.bWarningClearRequest := TRUE;
	        #nTriggerFailCount := 0;
	    ELSE
	        "DB_KeyenceCheckerIV3".aDev[#I_nID].Out.CommandControl.bWarningClearRequest := FALSE;
	    END_IF;
	    
	    //流程超时/Process over time
	    #tonProcessOvertime(IN := "DB_KeyenceCheckerIV3".aDev[#I_nID].Common.nMode <> #MODE_CHECKER_IDLE,
	                        PT := "DB_KeyenceCheckerIV3".aDev[#I_nID].Common.tMaxProcessTime);
	    IF #tonProcessOvertime.Q
	    THEN
	        "DB_KeyenceCheckerIV3".aDev[#I_nID].Common.nErrorNo := 1;
	    END_IF;
	    
	    //安全互锁/Safety interlock
	    IF NOT "DB_KeyenceCheckerIV3".aDev[#I_nID].Common.bEnable AND
	        "DB_KeyenceCheckerIV3".aDev[#I_nID].Common.nMode <> #MODE_CHECKER_IDLE
	    THEN
	        "DB_KeyenceCheckerIV3".aDev[#I_nID].Common.nErrorNo := 2;
	    END_IF;
	    
	    //模式无效/Mode invalid
	    //"DB_KeyenceCheckerIV2".aDev[#I_nID].Common.nErrorNo := 3;
	    
	    //相机警报/Vision warning
	    IF "DB_KeyenceCheckerIV3".aDev[#I_nID].In.CommandStatus.bWarning
	    THEN
	        "DB_KeyenceCheckerIV3".aDev[#I_nID].Common.nErrorNo := 6;
	    END_IF;
	    
	    //相机错误/Vision error
	    IF "DB_KeyenceCheckerIV3".aDev[#I_nID].In.CommandStatus.bError
	    THEN
	        "DB_KeyenceCheckerIV3".aDev[#I_nID].Common.nErrorNo := 7;
	    END_IF;
	    
	    //缓存溢出/Buffer overrun
	    IF "DB_KeyenceCheckerIV3".aDev[#I_nID].In.CommandStatus.bBufferOverrun
	    THEN
	        "DB_KeyenceCheckerIV3".aDev[#I_nID].Common.nErrorNo := 8;
	    END_IF;
	    
	    //程序切换失败/Program switching failed
	    IF "DB_KeyenceCheckerIV3".aDev[#I_nID].In.CommandStatus.bProgramSwitchingFailed
	    THEN
	        "DB_KeyenceCheckerIV3".aDev[#I_nID].Common.nErrorNo := 9;
	    END_IF;
	    
	    //触发失败/Trigger failed
	    IF #nTriggerFailCount >= 3
	    THEN
	        "DB_KeyenceCheckerIV3".aDev[#I_nID].Common.nErrorNo := 10;
	    END_IF;
	    
	    //外部主控注册图像失败/Master image registration failed
	    IF "DB_KeyenceCheckerIV3".aDev[#I_nID].In.CommandStatus.bMasterImageRegistrationFailed
	    THEN
	        "DB_KeyenceCheckerIV3".aDev[#I_nID].Common.nErrorNo := 11;
	    END_IF;
	    
	    //设定值更改失败/Setting value change failed
	    IF "DB_KeyenceCheckerIV3".aDev[#I_nID].In.CommandStatus.bChangeParameterFailed
	    THEN
	        "DB_KeyenceCheckerIV3".aDev[#I_nID].Common.nErrorNo := 12;
	    END_IF;
	    
	    //错误标志/Error flag
	    IF "DB_KeyenceCheckerIV3".aDev[#I_nID].Common.nErrorNo <> 0 THEN
	        "DB_KeyenceCheckerIV3".aDev[#I_nID].Common.nMode := #MODE_CHECKER_IDLE;
	        "DB_KeyenceCheckerIV3".aDev[#I_nID].Common.bError := TRUE;
	    END_IF;
	END_REGION
	
	REGION WarningMessages()
	    //************************************************************************************************
	    //警告信息/Warning messages
	    //************************************************************************************************
	    //复位警告信息/Reset warning messages
	    "DB_KeyenceCheckerIV3".aDev[#I_nID].Common.nWarningNo := 0;
	    
	    //警告/Warning flag
	    "DB_KeyenceCheckerIV3".aDev[#I_nID].Common.bWarning :=
	    "DB_KeyenceCheckerIV3".aDev[#I_nID].Common.nWarningNo <> 0;
	END_REGION
	
	REGION FrontGenaralControl()
	    //************************************************************************************************
	    //前端通用控制/Front genaral control
	    //************************************************************************************************
	    "DB_KeyenceCheckerIV3".aDev[#I_nID].Out.CommandControl.nProgramNo := "DB_KeyenceCheckerIV3".aDev[#I_nID].Para.nProgramNo;
	    
	    //结果更新完成标志位/Complete toggle sign
	    #rtrigCompleteToggle(CLK := "DB_KeyenceCheckerIV3".aDev[#I_nID].In.CommandStatus.bResultUpdateComplete);
	    #ftrigCompleteToggle(CLK := "DB_KeyenceCheckerIV3".aDev[#I_nID].In.CommandStatus.bResultUpdateComplete);
	    IF #rtrigCompleteToggle.Q OR #ftrigCompleteToggle.Q THEN
	        #bCompleteToggleSign := TRUE;
	    END_IF;
	END_REGION
	
	REGION AutoProcess()
	    //************************************************************************************************
	    //自动流程/Auto process
	    //************************************************************************************************
	    IF "DB_KeyenceCheckerIV3".aDev[#I_nID].Common.nMode <> #MODE_CHECKER_IDLE THEN
	        CASE #nStep OF
	                //******************************************************************************
	            0: //等待模式选择/Wait for mode selected
	                //设置下一个步号/Set next step
	                CASE "DB_KeyenceCheckerIV3".aDev[#I_nID].Common.nMode OF
	                    #MODE_CHECKER_START://开始相机/Start vision
	                        #nNextStep := 100;
	                        // #MODE_CHECKER_REGISTER://程序切换/Program switching
	                        //     #nNextStep := 200;
	                    #MODE_CHECKER_CLEAR://统计数据清除/Stastics Reset
	                        #nNextStep := 300;
	                    #MODE_CHECKER_RESET://初始化/Reset paramaters
	                        #nNextStep := 900;
	                    ELSE
	                        "DB_KeyenceCheckerIV3".aDev[#I_nID].Common.nErrorNo := 3;//模式无效/Mode invalid
	                END_CASE;
	                //复位流程完成标志/Reset done
	                "DB_KeyenceCheckerIV3".aDev[#I_nID].Common.bDone := FALSE;
	                #fbNextstep(I_bEnable := TRUE,
	                            I_bSeqMode := true,
	                            I_tTimeValue := t#0ms);
	                IF #fbNextstep.O_bStart THEN
	                    #nLastStep := #nStep;
	                    #nStep := #nNextStep;
	                END_IF;
	                //*************************************************************************************
	            100://检查程序号/Check program number
	                //设置下一个步号/Set next step
	                //
	                #bCompleteToggleSign := FALSE;
	                "DB_KeyenceCheckerIV3".aDev[#I_nID].Para.bProductOverallOK := FALSE;
	                "DB_KeyenceCheckerIV3".aDev[#I_nID].Para.bProductOverallNG := FALSE;
	                "DB_KeyenceCheckerIV3".aDev[#I_nID].Para.aToolResult := #aToolResultReset;
	                "DB_KeyenceCheckerIV3".aDev[#I_nID].Para.ToolResult := #ToolResultResult;
	                IF "DB_KeyenceCheckerIV3".aDev[#I_nID].In."DeviceStatus".nCurrentProgramNo <> "DB_KeyenceCheckerIV3".aDev[#I_nID].Out.CommandControl.nProgramNo
	                THEN
	                    #nNextStep := 110;
	                ELSE
	                    #nNextStep := 120;
	                END_IF;
	                //Condition
	                #bCondition := "DB_KeyenceCheckerIV3".aDev[#I_nID].In.CommandStatus.bRun AND NOT "DB_KeyenceCheckerIV3".aDev[#I_nID].In.CommandStatus.bBusy;
	                //Goto next step
	                #fbNextstep(I_bEnable := #bCondition,
	                            I_bSeqMode := true,
	                            I_tTimeValue := t#0ms);
	                IF #fbNextstep.O_bStart THEN
	                    #nLastStep := #nStep;
	                    #nStep := #nNextStep;
	                END_IF;
	                //*************************************************************************************
	            110://程序切换/Program switching
	                //设置下一个步号/Set next step
	                #nNextStep := 120;
	                //Action
	                "DB_KeyenceCheckerIV3".aDev[#I_nID].Out.CommandControl.bProgramSwitchingRequest := TRUE;
	                //Condition
	                #bCondition := "DB_KeyenceCheckerIV3".aDev[#I_nID].In.CommandStatus.bProgramSwitchingResponse AND NOT "DB_KeyenceCheckerIV3".aDev[#I_nID].In.CommandStatus.bProgramSwitchingFailed
	                AND "DB_KeyenceCheckerIV3".aDev[#I_nID].In."DeviceStatus".nCurrentProgramNo = "DB_KeyenceCheckerIV3".aDev[#I_nID].Out.CommandControl.nProgramNo;
	                //Goto next step
	                #fbNextstep(I_bEnable := #bCondition,
	                            I_bSeqMode := true,
	                            I_tTimeValue := t#0ms);
	                IF #fbNextstep.O_bStart THEN
	                    #nLastStep := #nStep;
	                    #nStep := #nNextStep;
	                    //复位程序选择/Reset program switch
	                    "DB_KeyenceCheckerIV3".aDev[#I_nID].Out.CommandControl.bProgramSwitchingRequest := FALSE;
	                END_IF;
	                //*************************************************************************************
	            120://触发输入/Trigger input 
	                //设置下一个步号/Set next step
	                IF "DB_KeyenceCheckerIV3".aDev[#I_nID].In.CommandStatus.bTriggerFailed THEN
	                    #nNextStep := 100;
	                    #nTriggerFailCount := #nTriggerFailCount + 1;
	                ELSE
	                    #nNextStep := 130;
	                    #nTriggerFailCount := 0;
	                END_IF;
	                //Action
	               // #bCompleteToggleSign := FALSE;
	                "DB_KeyenceCheckerIV3".aDev[#I_nID].Out.CommandControl.bTriggerRequest := TRUE;
	                //Condition
	                #bCondition := "DB_KeyenceCheckerIV3".aDev[#I_nID].In.CommandStatus.bTriggerResponse;
	                //Goto next step
	                #fbNextstep(I_bEnable := #bCondition,
	                            I_bSeqMode := true,
	                            I_tTimeValue := t#0ms);
	                IF #fbNextstep.O_bStart THEN
	                    #nLastStep := #nStep;
	                    #nStep := #nNextStep;
	                    //触发复位/Reset trigger 
	                    "DB_KeyenceCheckerIV3".aDev[#I_nID].Out.CommandControl.bTriggerRequest := FALSE;
	                END_IF;
	                //*************************************************************************************
	            130://等待结果判断/Waite for result 
	                //设置下一个步号/Set next step
	                #nNextStep := 0;
	                //Condition
	                #bCondition := NOT "DB_KeyenceCheckerIV3".aDev[#I_nID].In.CommandStatus.bBusy AND #bCompleteToggleSign;
	                //goto next step
	                #fbNextstep(I_bEnable := #bCondition,
	                            I_bSeqMode := true,
	                            I_tTimeValue := t#0ms);
	                IF #fbNextstep.O_bStart THEN
	                    #nLastStep := #nStep;
	                    #nStep := #nNextStep;
	                    //take result
	                    //Choose basic or extension tools
	                    FOR #nIndex3 := 1 TO 64 DO
	                        IF #nIndex3 <= 16 THEN
	                            "DB_KeyenceCheckerIV3".aDev[#I_nID].Para.aToolResult[#nIndex3] := "DB_KeyenceCheckerIV3".aDev[#I_nID].In.DeviceResults.aToolResult[#nIndex3];
	                        ELSE
	                            "DB_KeyenceCheckerIV3".aDev[#I_nID].Para.aToolResult[#nIndex3] := "DB_KeyenceCheckerIV3".aDev[#I_nID].In.ExtendedDeviceResult.aToolResult[#nIndex3];
	                        END_IF;
	                    END_FOR;
	                    "DB_KeyenceCheckerIV3".aDev[#I_nID].Para.bProductOverallOK := "DB_KeyenceCheckerIV3".aDev[#I_nID].In.DeviceResults.bOverallJudgmentOK;
	                    "DB_KeyenceCheckerIV3".aDev[#I_nID].Para.bProductOverallNG := "DB_KeyenceCheckerIV3".aDev[#I_nID].In.DeviceResults.bOverallJudgmentNG;
	                    "DB_KeyenceCheckerIV3".aDev[#I_nID].Para.ToolResult := "DB_KeyenceCheckerIV3".aDev[#I_nID].In.ToolResult;
	                    "DB_KeyenceCheckerIV3".aDev[#I_nID].Common.bDone := TRUE;
	                    "DB_KeyenceCheckerIV3".aDev[#I_nID].Common.nMode := #MODE_CHECKER_IDLE;
	                END_IF;
	                //*************************************************************************************
	                // 200: //检查程序号/Check program number
	                //     //设置下一个步号/Set next step
	                //     IF "DB_KeyenceCheckerIV2".aDev[#I_nID].In."DeviceStatus".nCurrentProgramNo <> "DB_KeyenceCheckerIV2".aDev[#I_nID].Out.CommandControl.nProgramNo
	                //     THEN
	                //         #nNextStep := 210;
	                //     ELSE
	                //         #nNextStep := 220;
	                //     END_IF;
	                //     //Condition
	                //     #bCondition := "DB_KeyenceCheckerIV2".aDev[#I_nID].In.CommandStatus.bRun AND NOT "DB_KeyenceCheckerIV2".aDev[#I_nID].In.CommandStatus.bBusy;
	                //     //Goto next step
	                //     #fbNextstep(I_bEnable := #bCondition,
	                //                 I_bSeqMode := true,
	                //                 I_tTimeValue := t#0ms);
	                //     IF #fbNextstep.O_bStart THEN
	                //         #nLastStep := #nStep;
	                //         #nStep := #nNextStep;
	                //     END_IF;
	                //     //*************************************************************************************
	                // 210: //程序切换/Program switching
	                //     //设置下一个步号/Set next step
	                //     #nNextStep := 120;
	                //     //Action
	                //     "DB_KeyenceCheckerIV2".aDev[#I_nID].Out.CommandControl.bProgramSwitchingRequest := TRUE;
	                //     //Condition
	                //     #bCondition := "DB_KeyenceCheckerIV2".aDev[#I_nID].In.CommandStatus.bProgramSwitchingResponse AND NOT  "DB_KeyenceCheckerIV2".aDev[#I_nID].In.CommandStatus.bProgramSwitchingFailed
	                //     AND "DB_KeyenceCheckerIV2".aDev[#I_nID].In."DeviceStatus".nCurrentProgramNo = "DB_KeyenceCheckerIV2".aDev[#I_nID].Out.CommandControl.nProgramNo;
	                //     //Goto next step
	                //     #fbNextstep(I_bEnable := #bCondition,
	                //                 I_bSeqMode := true,
	                //                 I_tTimeValue := t#0ms);
	                //     IF #fbNextstep.O_bStart THEN
	                //         #nLastStep := #nStep;
	                //         #nStep := #nNextStep;
	                //         //复位程序选择/Reset program switch
	                //         "DB_KeyenceCheckerIV2".aDev[#I_nID].Out.CommandControl.bProgramSwitchingRequest := FALSE;
	                //     END_IF;
	                //     //*************************************************************************************
	                // 220: //外部主控注册图像/Registering a master image externally
	                //     //设置下一个步号/Set next step
	                //     #nNextStep := 0;
	                //     //Action
	                //     "DB_KeyenceCheckerIV2".aDev[#I_nID].Out.CommandControl.bMasterRegistrationRequest := TRUE;
	                //     //Condition
	                //     #bCondition := "DB_KeyenceCheckerIV2".aDev[#I_nID].In.CommandStatus.bMasterImageRegistration AND NOT "DB_KeyenceCheckerIV2".aDev[#I_nID].In.CommandStatus.bBusy
	                //     AND NOT "DB_KeyenceCheckerIV2".aDev[#I_nID].In.CommandStatus.bMasterImageRegistrationFailed;
	                //     //Goto next step
	                //     #fbNextstep(I_bEnable := #bCondition,
	                //                 I_bSeqMode := true,
	                //                 I_tTimeValue := t#0ms);
	                //     IF #fbNextstep.O_bStart THEN
	                //         #nLastStep := #nStep;
	                //         #nStep := #nNextStep;
	                //         //Reset process
	                //         "DB_KeyenceCheckerIV2".aDev[#I_nID].Out.CommandControl.bMasterRegistrationRequest := FALSE;
	                //         //Set process done
	                //         "DB_KeyenceCheckerIV2".aDev[#I_nID].Common.bDone := TRUE;
	                //         "DB_KeyenceCheckerIV2".aDev[#I_nID].Common.nMode := #MODE_CHECKER_IDLE;
	                //     END_IF;
	                //*************************************************************************************
	            300: //等待相机准备完成/Wait Camera ready
	                //设置下一个步号/Set next step
	                #nNextStep := 310;
	                //Condition
	                #bCondition := "DB_KeyenceCheckerIV3".aDev[#I_nID].In.CommandStatus.bRun AND NOT "DB_KeyenceCheckerIV3".aDev[#I_nID].In.CommandStatus.bBusy;
	                //Goto next step
	                #fbNextstep(I_bEnable := #bCondition,
	                            I_bSeqMode := true,
	                            I_tTimeValue := t#0ms);
	                IF #fbNextstep.O_bStart THEN
	                    #nLastStep := #nStep;
	                    #nStep := #nNextStep;
	                END_IF;
	                //*************************************************************************************
	            310: //统计数据清除/Stastics reset
	                //设置下一个步号/Set next step
	                #nNextStep := 0;
	                //Action
	                "DB_KeyenceCheckerIV3".aDev[#I_nID].Out.CommandControl.bStatisticsResetRequest := TRUE;
	                //Condition
	                #bCondition := "DB_KeyenceCheckerIV3".aDev[#I_nID].In.CommandStatus.bStatisticsResetResponse;
	                //Goto next step
	                #fbNextstep(I_bEnable := #bCondition,
	                            I_bSeqMode := true,
	                            I_tTimeValue := t#0ms);
	                IF #fbNextstep.O_bStart THEN
	                    #nLastStep := #nStep;
	                    #nStep := #nNextStep;
	                    //停止统计数据清楚/Stop stastics reset
	                    "DB_KeyenceCheckerIV3".aDev[#I_nID].Out.CommandControl.bStatisticsResetRequest := FALSE;
	                    //动作完成/Action Done
	                    "DB_KeyenceCheckerIV3".aDev[#I_nID].Common.bDone := TRUE;
	                    "DB_KeyenceCheckerIV3".aDev[#I_nID].Common.nMode := #MODE_CHECKER_IDLE;
	                END_IF;
	                //*************************************************************************************
	            900: //等待相机准备完成/Wait Camera ready
	                //设置下一个步号/Set next step
	                #nNextStep := 910;
	                //Condition
	                #bCondition := "DB_KeyenceCheckerIV3".aDev[#I_nID].In.CommandStatus.bRun AND NOT "DB_KeyenceCheckerIV3".aDev[#I_nID].In.CommandStatus.bBusy;
	                //Goto next step
	                #fbNextstep(I_bEnable := #bCondition,
	                            I_bSeqMode := true,
	                            I_tTimeValue := t#0ms);
	                IF #fbNextstep.O_bStart THEN
	                    #nLastStep := #nStep;
	                    #nStep := #nNextStep;
	                END_IF;
	                //*************************************************************************************
	            910: //初始化/Reset paramaters
	                //设置下一个步号/Set next step
	                #nNextStep := 0;
	                //Action
	                //清除PLC数据/Reset PLC data
	                #nTriggerFailCount := 0;
	                "DB_KeyenceCheckerIV3".aDev[#I_nID].Out.CommandControl.bTriggerRequest := FALSE;
	                "DB_KeyenceCheckerIV3".aDev[#I_nID].Out.CommandControl.bMasterRegistrationRequest := FALSE;
	                "DB_KeyenceCheckerIV3".aDev[#I_nID].Out.CommandControl.bProgramSwitchingRequest := FALSE;
	                "DB_KeyenceCheckerIV3".aDev[#I_nID].Out.CommandControl.bParameterChangeRequest := FALSE;
	                "DB_KeyenceCheckerIV3".aDev[#I_nID].Out.CommandControl.bResultAcquisitionCompleteNotification := FALSE;
	                "DB_KeyenceCheckerIV3".aDev[#I_nID].Para.bProductOverallOK := FALSE;
	                "DB_KeyenceCheckerIV3".aDev[#I_nID].Para.bProductOverallNG := FALSE;
	                "DB_KeyenceCheckerIV3".aDev[#I_nID].Para.aToolResult := #aToolResultReset;
	                "DB_KeyenceCheckerIV3".aDev[#I_nID].Para.ToolResult := #ToolResultResult;
	                //清除缓存结果/Reset buffer 
	                "DB_KeyenceCheckerIV3".aDev[#I_nID].Out.CommandControl.bBufferClearRequest := TRUE;
	                //清除统计数据/Reset Stastics
	                "DB_KeyenceCheckerIV3".aDev[#I_nID].Out.CommandControl.bStatisticsResetRequest := TRUE;
	                //condition
	                #bCondition := "DB_KeyenceCheckerIV3".aDev[#I_nID].In.CommandStatus.bBufferClearResponse AND "DB_KeyenceCheckerIV3".aDev[#I_nID].In.CommandStatus.bStatisticsResetResponse;
	                //goto next step
	                #fbNextstep(I_bEnable := #bCondition,
	                            I_bSeqMode := true,
	                            I_tTimeValue := t#0ms);
	                IF #fbNextstep.O_bStart THEN
	                    #nLastStep := #nStep;
	                    #nStep := #nNextStep;
	                    //初始化请求停止/Stop reset
	                    "DB_KeyenceCheckerIV3".aDev[#I_nID].Out.CommandControl.bBufferClearRequest := FALSE;
	                    "DB_KeyenceCheckerIV3".aDev[#I_nID].Out.CommandControl.bStatisticsResetRequest := FALSE;
	                    //动作完成/Action Done
	                    "DB_KeyenceCheckerIV3".aDev[#I_nID].Common.bDone := TRUE;
	                    "DB_KeyenceCheckerIV3".aDev[#I_nID].Common.nMode := #MODE_CHECKER_IDLE;
	                END_IF;
	        END_CASE;
	    ELSE
	        #nStep := 0;
	        //Reset signals
	        "DB_KeyenceCheckerIV3".aDev[#I_nID].Out.CommandControl.bTriggerRequest := FALSE;
	        "DB_KeyenceCheckerIV3".aDev[#I_nID].Out.CommandControl.bMasterRegistrationRequest := FALSE;
	        "DB_KeyenceCheckerIV3".aDev[#I_nID].Out.CommandControl.bProgramSwitchingRequest := FALSE;
	        "DB_KeyenceCheckerIV3".aDev[#I_nID].Out.CommandControl.bParameterChangeRequest := FALSE;
	        "DB_KeyenceCheckerIV3".aDev[#I_nID].Out.CommandControl.bResultAcquisitionCompleteNotification := FALSE;
	        "DB_KeyenceCheckerIV3".aDev[#I_nID].Out.CommandControl.bBufferClearRequest := FALSE;
	        "DB_KeyenceCheckerIV3".aDev[#I_nID].Out.CommandControl.bStatisticsResetRequest := FALSE;
	        #bCompleteToggleSign := FALSE;
	        #bCondition := FALSE;
	        #fbNextstep(I_bEnable := #bCondition,
	                    I_bSeqMode := TRUE,
	                    I_tTimeValue := t#0ms);
	    END_IF;
	END_REGION
	
	REGION BehindGeneralControl()
	    //************************************************************************************************
	    //后端通用控制/Behind genaral control
	    //************************************************************************************************
	    //设备启动停止/Device mode control
	    #rtrigManualMode(CLK := "DB_KeyenceCheckerIV3".aDev[#I_nID].Common.nModeSwitch = "MS_MANUAL");
	    #ftrigManualMode(CLK := "DB_KeyenceCheckerIV3".aDev[#I_nID].Common.nModeSwitch = "MS_MANUAL");
	    IF "DB_KeyenceCheckerIV3".aDev[#I_nID].Common.nModeSwitch = "MS_EMPTY" OR
	        #rtrigManualMode.Q OR #ftrigManualMode.Q
	    THEN
	        "DB_KeyenceCheckerIV3".aDev[#I_nID].Common.nMode := #MODE_CHECKER_IDLE;
	    END_IF;
	    //触摸屏显示工具结果/Tool result to HMI
	    FOR #nIdx := 1 TO 16 BY 1 DO
	        IF "DB_KeyenceCheckerIV3".aDev[#I_nID].Para.ToolResult[#nIdx].nToolMatchingRateMIN = 0 AND "DB_KeyenceCheckerIV3".aDev[#I_nID].Para.ToolResult[#nIdx].nToolMatchingRate = 0 THEN
	            //工具未使用/Tool is unuseful
	            "DB_KeyenceCheckerIV3".aDev[#I_nID].Para.aToolResultHMI[#nIdx] := 2;//灰色/Gray
	        ELSE
	            IF "DB_KeyenceCheckerIV3".aDev[#I_nID].Para.aToolResult[#nIdx] THEN
	                //工具结果OK/Tool result is OK
	                "DB_KeyenceCheckerIV3".aDev[#I_nID].Para.aToolResultHMI[#nIdx] := 1;//绿色/Green
	            END_IF;
	            IF NOT "DB_KeyenceCheckerIV3".aDev[#I_nID].Para.aToolResult[#nIdx] THEN
	                //工具结果NG/Tool result is NG
	                "DB_KeyenceCheckerIV3".aDev[#I_nID].Para.aToolResultHMI[#nIdx] := 0;//红色/Red
	            END_IF;
	        END_IF;
	    END_FOR;
	END_REGION
	
	REGION CopyWriteData()
	    //************************************************************************************************
	    //分配输出数据/Asignment of the output data (Controlword)
	    //************************************************************************************************
	    //指令控制/Command control Address 
	    //Address 0
	    #nByte.%X0 := "DB_KeyenceCheckerIV3".aDev[#I_nID].Out.CommandControl.bTriggerRequest;
	    #nByte.%X1 := "DB_KeyenceCheckerIV3".aDev[#I_nID].Out.CommandControl.bMasterRegistrationRequest;
	    #nByte.%X2 := "DB_KeyenceCheckerIV3".aDev[#I_nID].Out.CommandControl.bProgramSwitchingRequest;
	    #nByte.%X3 := "DB_KeyenceCheckerIV3".aDev[#I_nID].Out.CommandControl.bWarningClearRequest;
	    #nByte.%X4 := "DB_KeyenceCheckerIV3".aDev[#I_nID].Out.CommandControl.bStatisticsResetRequest;
	    #nByte.%X5 := "DB_KeyenceCheckerIV3".aDev[#I_nID].Out.CommandControl.bBufferClearRequest;
	    #nByte.%X6 := "DB_KeyenceCheckerIV3".aDev[#I_nID].Out.CommandControl.bSDCardSaveStopRequest;
	    #nByte.%X7 := "DB_KeyenceCheckerIV3".aDev[#I_nID].Out.CommandControl.bParameterChangeRequest;
	    #aOutput_Byte1[0] := #nByte;
	    //Aaddress 1
	    #nByte := "DB_KeyenceCheckerIV3".aDev[#I_nID].Out.CommandControl.nReserved1;
	    #aOutput_Byte1[1] := #nByte;
	    //Aaddress 2
	    #nByte.%X0 := "DB_KeyenceCheckerIV3".aDev[#I_nID].Out.CommandControl.bResultAcquisitionCompleteNotification;
	    #nByte.%X1 := "DB_KeyenceCheckerIV3".aDev[#I_nID].Out.CommandControl.bReserved2;
	    #nByte.%X2 := "DB_KeyenceCheckerIV3".aDev[#I_nID].Out.CommandControl.bReserved3;
	    #nByte.%X3 := "DB_KeyenceCheckerIV3".aDev[#I_nID].Out.CommandControl.bReserved4;
	    #nByte.%X4 := "DB_KeyenceCheckerIV3".aDev[#I_nID].Out.CommandControl.bReserved5;
	    #nByte.%X5 := "DB_KeyenceCheckerIV3".aDev[#I_nID].Out.CommandControl.bReserved6;
	    #nByte.%X6 := "DB_KeyenceCheckerIV3".aDev[#I_nID].Out.CommandControl.bReserved7;
	    #nByte.%X7 := "DB_KeyenceCheckerIV3".aDev[#I_nID].Out.CommandControl.bReserved8;
	    #aOutput_Byte1[2] := #nByte;
	    //Address 3 
	    #nByte := "DB_KeyenceCheckerIV3".aDev[#I_nID].Out.CommandControl.nReserved9;
	    #aOutput_Byte1[3] := #nByte;
	    //程序号/Program number
	    #nWord := "DB_KeyenceCheckerIV3".aDev[#I_nID].Out.CommandControl.nProgramNo;
	    #aOutput_Byte1[4] := #aWord[0];
	    #aOutput_Byte1[5] := #aWord[1];
	    //设定值设定编号/Setting value setting number
	    #nWord := "DB_KeyenceCheckerIV3".aDev[#I_nID].Out.CommandControl.nSetNumber;
	    #aOutput_Byte1[6] := #aWord[0];
	    #aOutput_Byte1[7] := #aWord[1];
	    //设定值/Setting value
	    #nDWord := "DB_KeyenceCheckerIV3".aDev[#I_nID].Out.CommandControl.nSetParameter;
	    #aOutput_Byte1[8] := #aDWord[0];
	    #aOutput_Byte1[9] := #aDWord[1];
	    #aOutput_Byte1[10] := #aDWord[2];
	    #aOutput_Byte1[11] := #aDWord[3];
	END_REGION
	
	REGION WriteData()
	    //************************************************************************************************ 
	    //向接口写入数据/Write data to interface
	    //************************************************************************************************ 
	    //指令控制/Command control
	    #aRetvalWrite[1] := DPWR_DAT(LADDR := "DB_KeyenceCheckerIV3".aDev[#I_nID].Para.nOutAdr1, RECORD := #aOutput_Byte1);
	END_REGION
	
	REGION Steps()
	    //************************************************************************************************ 
	    //步数显示在触摸屏/Steps show in HMI
	    //************************************************************************************************ 
	    "DB_KeyenceCheckerIV3".aDev[#I_nID].Common.nLastStep := #nLastStep;
	    "DB_KeyenceCheckerIV3".aDev[#I_nID].Common.nCurrentStep := #nStep;
	    "DB_KeyenceCheckerIV3".aDev[#I_nID].Common.nNextStep := #nNextStep;
	    
	    //流程时间/Process Time
	    IF "DB_KeyenceCheckerIV3".aDev[#I_nID].Common.nMode <> #MODE_CHECKER_IDLE
	    THEN
	        "DB_KeyenceCheckerIV3".aDev[#I_nID].Common.tActProcessTime := #tonProcessOvertime.ET;
	    END_IF;
	END_REGION
END_FUNCTION_BLOCK

FUNCTION_BLOCK "Axis_FB"
{ S7_Optimized_Access := 'FALSE' }
VERSION : 0.1
   VAR 
      IAI_Axis : Array[1..3] of "IAI_BASE_FB";
   END_VAR


BEGIN
	///Z轴
	#IAI_Axis[1]();
	
	#IAI_Axis[1].Axis_ID := 1;
	#IAI_Axis[1]."Input 4 word_Man1" := "OP10_384A1~Input_4_word_7";
	#IAI_Axis[1]."Input 4 word_Man2" := "OP10_384A1~Input_4_word_8";
	#IAI_Axis[1]."Input 4 word_1" := "OP10_384A1~Input_4_word_3";
	#IAI_Axis[1]."Input 4 word_2" := "OP10_384A1~Input_4_word_4";
	#IAI_Axis[1]."Output 4 word_Man1" := "OP10_384A1~Output_4_word_1";
	#IAI_Axis[1]."Output 4 word_Man2" := "OP10_384A1~Output_4_word_2";
	#IAI_Axis[1]."Output 4 word_1" := "OP10_384A1~Output_4_word_5";
	#IAI_Axis[1]."Output 4 word_2" := "OP10_384A1~Output_4_word_6";
	
	#IAI_Axis[1].Mode:= "ModeDB".Gen;
	#IAI_Axis[1].Par.PositionWidth := 0.05;
	#IAI_Axis[1].Par.AccSpeed := 10;
	#IAI_Axis[1].Par."Limt+Pos" := 362000.0;
	#IAI_Axis[1].Par."Limt-Pos" := -30000.0;
	#IAI_Axis[1].Interfere := TRUE;
	#IAI_Axis[1].RunSetTime := T#20S;
	#IAI_Axis[1].Par.GoPosInterfere[0] := TRUE;
	#IAI_Axis[1].Par.GoPosInterfere[1] := TRUE;
	#IAI_Axis[1].Par.GoPosInterfere[2] := TRUE;
	#IAI_Axis[1].Par.GoPosInterfere[3] := TRUE;
	#IAI_Axis[1].Par.GoPosInterfere[4] := TRUE;
	#IAI_Axis[1].Par.GoPosInterfere[5] := TRUE;
	#IAI_Axis[1].AutoPointStart := "IAI_A1".In.iAutoStart;
	
	"IAI_A1".Auto.Pos[1].Pos:=#IAI_Axis[1].Par.TargetPosition[1] := "Parameter".AxisRun.Axis[5].Pos1.Position;
	"IAI_A1".Auto.Pos[1].Vel :=#IAI_Axis[1].Par.TargetSpeed[1] := "Parameter".AxisRun.Axis[5].Pos1.Speed;
	
	"IAI_A1".Auto.Pos[2].Pos:=#IAI_Axis[1].Par.TargetPosition[2] := "Parameter".AxisRun.Axis[5].Pos2.Position;
	"IAI_A1".Auto.Pos[2].Vel :=#IAI_Axis[1].Par.TargetSpeed[2] := "Parameter".AxisRun.Axis[5].Pos2.Speed;
	
	"IAI_A1".Auto.Pos[3].Pos:=#IAI_Axis[1].Par.TargetPosition[3] := "Parameter".AxisRun.Axis[5].Pos3.Position;
	"IAI_A1".Auto.Pos[3].Vel :=#IAI_Axis[1].Par.TargetSpeed[3] := "Parameter".AxisRun.Axis[5].Pos3.Speed;
	
	"IAI_A1".Auto.Pos[4].Pos:=#IAI_Axis[1].Par.TargetPosition[4] := "Parameter".AxisRun.Axis[5].Pos4.Position;
	"IAI_A1".Auto.Pos[4].Vel :=#IAI_Axis[1].Par.TargetSpeed[4] := "Parameter".AxisRun.Axis[5].Pos4.Speed;
	
	"IAI_A1".Auto.Pos[5].Pos:=#IAI_Axis[1].Par.TargetPosition[5] := "Parameter".AxisRun.Axis[5].Pos5.Position;
	"IAI_A1".Auto.Pos[5].Vel :=#IAI_Axis[1].Par.TargetSpeed[5] := "Parameter".AxisRun.Axis[5].Pos5.Speed;
	
	"IAI_A1".Auto.Pos[6].Pos := #IAI_Axis[1].Par.TargetPosition[6] := "Parameter".AxisRun.Axis[5].Pos6.Position;
	"IAI_A1".Auto.Pos[6].Vel := #IAI_Axis[1].Par.TargetSpeed[6] := "Parameter".AxisRun.Axis[5].Pos6.Speed;
	
	"IAI_A1".Auto.Pos[7].Pos := #IAI_Axis[1].Par.TargetPosition[7] := "Parameter".AxisRun.Axis[5].Pos7.Position;
	"IAI_A1".Auto.Pos[7].Vel := #IAI_Axis[1].Par.TargetSpeed[7] := "Parameter".AxisRun.Axis[5].Pos7.Speed;
	
	"IAI_A1".Auto.Pos[8].Pos := #IAI_Axis[1].Par.TargetPosition[8] := "Parameter".AxisRun.Axis[5].Pos8.Position;
	"IAI_A1".Auto.Pos[8].Vel := #IAI_Axis[1].Par.TargetSpeed[8] := "Parameter".AxisRun.Axis[5].Pos8.Speed;
	
	"IAI_A1".Auto.Pos[9].Pos := #IAI_Axis[1].Par.TargetPosition[9] := "Parameter".AxisRun.Axis[5].Pos6.Position-4.0;
	"IAI_A1".Auto.Pos[9].Vel := #IAI_Axis[1].Par.TargetSpeed[9] := "Parameter".AxisRun.Axis[5].Pos6.Speed;
	
	"IAI_A1".Auto.Pos[10].Pos := #IAI_Axis[1].Par.TargetPosition[10] := "Parameter".AxisRun.Axis[5].Pos10.Position;
	"IAI_A1".Auto.Pos[10].Vel := #IAI_Axis[1].Par.TargetSpeed[10] := "Parameter".AxisRun.Axis[5].Pos10.Speed;
	
	//X轴
	#IAI_Axis[2]();
	
	#IAI_Axis[2].Axis_ID := 2;
	#IAI_Axis[2]."Input 4 word_Man1" := "OP10_384A1~Input_4_word_7";
	#IAI_Axis[2]."Input 4 word_Man2" := "OP10_384A1~Input_4_word_8";
	#IAI_Axis[2]."Input 4 word_1" := "OP10_384A1~Input_4_word_5";
	#IAI_Axis[2]."Input 4 word_2" := "OP10_384A1~Input_4_word_6";
	#IAI_Axis[2]."Output 4 word_Man1" := "OP10_384A1~Output_4_word_1";
	#IAI_Axis[2]."Output 4 word_Man2" := "OP10_384A1~Output_4_word_2";
	#IAI_Axis[2]."Output 4 word_1" := "OP10_384A1~Output_4_word_7";
	#IAI_Axis[2]."Output 4 word_2" := "OP10_384A1~Output_4_word_8";
	
	#IAI_Axis[2].Mode := "ModeDB".Gen;
	#IAI_Axis[2].Par.PositionWidth := 0.05;
	#IAI_Axis[2].Par.AccSpeed := 10;
	#IAI_Axis[2].Par."Limt+Pos" := 362000.0;
	#IAI_Axis[2].Par."Limt-Pos" := -30000.0;
	#IAI_Axis[2].Interfere := TRUE;
	#IAI_Axis[2].RunSetTime := T#20S; 
	#IAI_Axis[2].Par.GoPosInterfere[0] := TRUE;
	#IAI_Axis[2].Par.GoPosInterfere[1] := TRUE;
	#IAI_Axis[2].Par.GoPosInterfere[2] := TRUE;
	#IAI_Axis[2].Par.GoPosInterfere[3] := TRUE;
	#IAI_Axis[2].Par.GoPosInterfere[4] := TRUE;
	#IAI_Axis[2].Par.GoPosInterfere[5] := TRUE;
	#IAI_Axis[2].AutoPointStart := "IAI_A2".In.iAutoStart;
	
	"IAI_A2".Auto.Pos[1].Pos:=#IAI_Axis[2].Par.TargetPosition[1] := "Parameter".AxisRun.Axis[6].Pos1.Position;
	"IAI_A2".Auto.Pos[1].Vel := #IAI_Axis[2].Par.TargetSpeed[1] := "Parameter".AxisRun.Axis[6].Pos1.Speed;
	
	"IAI_A2".Auto.Pos[2].Pos:=#IAI_Axis[2].Par.TargetPosition[2] := "Parameter".AxisRun.Axis[6].Pos2.Position;
	"IAI_A2".Auto.Pos[2].Vel :=#IAI_Axis[2].Par.TargetSpeed[2] := "Parameter".AxisRun.Axis[6].Pos2.Speed;
	
	"IAI_A2".Auto.Pos[3].Pos:=#IAI_Axis[2].Par.TargetPosition[3] := "Parameter".AxisRun.Axis[6].Pos3.Position;
	"IAI_A2".Auto.Pos[3].Vel :=#IAI_Axis[2].Par.TargetSpeed[3] := "Parameter".AxisRun.Axis[6].Pos3.Speed;
	
	"IAI_A2".Auto.Pos[4].Pos:=#IAI_Axis[2].Par.TargetPosition[4] := "Parameter".AxisRun.Axis[6].Pos4.Position;
	"IAI_A2".Auto.Pos[4].Vel :=#IAI_Axis[2].Par.TargetSpeed[4] := "Parameter".AxisRun.Axis[6].Pos4.Speed;
	
	"IAI_A2".Auto.Pos[5].Pos:=#IAI_Axis[2].Par.TargetPosition[5] := "Parameter".AxisRun.Axis[6].Pos5.Position;
	"IAI_A2".Auto.Pos[5].Vel :=#IAI_Axis[2].Par.TargetSpeed[5] := "Parameter".AxisRun.Axis[6].Pos5.Speed;
	
	"IAI_A2".Auto.Pos[6].Pos := #IAI_Axis[2].Par.TargetPosition[6] := "Parameter".AxisRun.Axis[6].Pos6.Position;
	"IAI_A2".Auto.Pos[6].Vel := #IAI_Axis[2].Par.TargetSpeed[6] := "Parameter".AxisRun.Axis[6].Pos6.Speed;
	
	"IAI_A2".Auto.Pos[7].Pos := #IAI_Axis[2].Par.TargetPosition[7] := "Parameter".AxisRun.Axis[6].Pos7.Position;
	"IAI_A2".Auto.Pos[7].Vel := #IAI_Axis[2].Par.TargetSpeed[7] := "Parameter".AxisRun.Axis[6].Pos7.Speed;
	
	"IAI_A2".Auto.Pos[8].Pos := #IAI_Axis[2].Par.TargetPosition[8] := "Parameter".AxisRun.Axis[6].Pos8.Position;
	"IAI_A2".Auto.Pos[8].Vel := #IAI_Axis[2].Par.TargetSpeed[8] := "Parameter".AxisRun.Axis[6].Pos8.Speed;
	
	"IAI_A2".Auto.Pos[9].Pos := #IAI_Axis[2].Par.TargetPosition[9] := "Parameter".AxisRun.Axis[6].Pos9.Position;
	"IAI_A2".Auto.Pos[9].Vel := #IAI_Axis[2].Par.TargetSpeed[9] := "Parameter".AxisRun.Axis[6].Pos9.Speed;
	
	"IAI_A2".Auto.Pos[10].Pos := #IAI_Axis[2].Par.TargetPosition[10] := "Parameter".AxisRun.Axis[6].Pos10.Position;
	"IAI_A2".Auto.Pos[10].Vel := #IAI_Axis[2].Par.TargetSpeed[10] := "Parameter".AxisRun.Axis[6].Pos10.Speed;
	
	///Y轴
	#IAI_Axis[3]();
	
	#IAI_Axis[3].Axis_ID := 3;
	#IAI_Axis[3]."Input 4 word_Man1" := "OP10_384A1~Input_4_word_7";
	#IAI_Axis[3]."Input 4 word_Man2" := "OP10_384A1~Input_4_word_8";
	#IAI_Axis[3]."Input 4 word_1" := "OP10_384A1~Input_4_word_1";
	#IAI_Axis[3]."Input 4 word_2" := "OP10_384A1~Input_4_word_2";
	#IAI_Axis[3]."Output 4 word_Man1" := "OP10_384A1~Output_4_word_1";
	#IAI_Axis[3]."Output 4 word_Man2" := "OP10_384A1~Output_4_word_2";
	#IAI_Axis[3]."Output 4 word_1" := "OP10_384A1~Output_4_word_3";
	#IAI_Axis[3]."Output 4 word_2" := "OP10_384A1~Output_4_word_4";
	
	#IAI_Axis[3].Mode := "ModeDB".Gen;
	#IAI_Axis[3].Par.PositionWidth := 0.05;
	#IAI_Axis[3].Par.AccSpeed := 10;
	#IAI_Axis[3].Par."Limt+Pos" := 362000.0;
	#IAI_Axis[3].Par."Limt-Pos" := -30000.0;
	#IAI_Axis[3].Interfere := TRUE;
	#IAI_Axis[3].RunSetTime := T#20S;
	#IAI_Axis[3].Par.GoPosInterfere[0] := TRUE;
	#IAI_Axis[3].Par.GoPosInterfere[1] := TRUE;
	#IAI_Axis[3].Par.GoPosInterfere[2] := TRUE;
	#IAI_Axis[3].Par.GoPosInterfere[3] := TRUE;
	#IAI_Axis[3].Par.GoPosInterfere[4] := TRUE;
	#IAI_Axis[3].Par.GoPosInterfere[5] := TRUE;
	#IAI_Axis[3].AutoPointStart := "IAI_A3".In.iAutoStart;
	
	"IAI_A3".Auto.Pos[1].Pos:=#IAI_Axis[3].Par.TargetPosition[1] := "Parameter".AxisRun.Axis[7].Pos1.Position;
	"IAI_A3".Auto.Pos[1].Vel :=#IAI_Axis[3].Par.TargetSpeed[1] := "Parameter".AxisRun.Axis[7].Pos1.Speed;
	
	"IAI_A3".Auto.Pos[2].Pos:=#IAI_Axis[3].Par.TargetPosition[2] := "Parameter".AxisRun.Axis[7].Pos2.Position;
	"IAI_A3".Auto.Pos[2].Vel :=#IAI_Axis[3].Par.TargetSpeed[2] := "Parameter".AxisRun.Axis[7].Pos2.Speed;
	
	"IAI_A3".Auto.Pos[3].Pos:=#IAI_Axis[3].Par.TargetPosition[3] := "Parameter".AxisRun.Axis[7].Pos3.Position;
	"IAI_A3".Auto.Pos[3].Vel :=#IAI_Axis[3].Par.TargetSpeed[3] := "Parameter".AxisRun.Axis[7].Pos3.Speed;
	
	"IAI_A3".Auto.Pos[4].Pos:=#IAI_Axis[3].Par.TargetPosition[4] := "Parameter".AxisRun.Axis[7].Pos4.Position;
	"IAI_A3".Auto.Pos[4].Vel :=#IAI_Axis[3].Par.TargetSpeed[4] := "Parameter".AxisRun.Axis[7].Pos4.Speed;
	
	"IAI_A3".Auto.Pos[5].Pos:=#IAI_Axis[3].Par.TargetPosition[5] := "Parameter".AxisRun.Axis[7].Pos5.Position;
	"IAI_A3".Auto.Pos[5].Vel :=#IAI_Axis[3].Par.TargetSpeed[5] := "Parameter".AxisRun.Axis[7].Pos5.Speed;
	
	"IAI_A3".Auto.Pos[6].Pos := #IAI_Axis[3].Par.TargetPosition[6] := "Parameter".AxisRun.Axis[7].Pos6.Position;
	"IAI_A3".Auto.Pos[6].Vel := #IAI_Axis[3].Par.TargetSpeed[6] := "Parameter".AxisRun.Axis[7].Pos6.Speed;
	
	"IAI_A3".Auto.Pos[7].Pos := #IAI_Axis[3].Par.TargetPosition[7] := "Parameter".AxisRun.Axis[7].Pos7.Position;
	"IAI_A3".Auto.Pos[7].Vel := #IAI_Axis[3].Par.TargetSpeed[7] := "Parameter".AxisRun.Axis[7].Pos7.Speed;
	
	"IAI_A3".Auto.Pos[8].Pos := #IAI_Axis[3].Par.TargetPosition[8] := "Parameter".AxisRun.Axis[7].Pos8.Position;
	"IAI_A3".Auto.Pos[8].Vel := #IAI_Axis[3].Par.TargetSpeed[8] := "Parameter".AxisRun.Axis[7].Pos8.Speed;
	
	"IAI_A3".Auto.Pos[9].Pos := #IAI_Axis[3].Par.TargetPosition[9] := "Parameter".AxisRun.Axis[7].Pos9.Position;
	"IAI_A3".Auto.Pos[9].Vel := #IAI_Axis[3].Par.TargetSpeed[9] := "Parameter".AxisRun.Axis[7].Pos9.Speed;
	
	"IAI_A3".Auto.Pos[10].Pos := #IAI_Axis[3].Par.TargetPosition[10] := "Parameter".AxisRun.Axis[7].Pos10.Position;
	"IAI_A3".Auto.Pos[10].Vel := #IAI_Axis[3].Par.TargetSpeed[10] := "Parameter".AxisRun.Axis[7].Pos10.Speed;
	
	/////////////////HNI_DATA_PUT&GET////////
	IF "ModeDB".Gen.Out.Manual THEN
	    #IAI_Axis["HMISystemDB".HMI_Axis.INPUT.Axis_ID].Par.Speed := "HMISystemDB".HMI_Axis.INPUT.Speed;
	    #IAI_Axis["HMISystemDB".HMI_Axis.INPUT.Axis_ID].Par.SimplyTrigger := "HMISystemDB".HMI_Axis.INPUT.SimplyTrigger;
	    #IAI_Axis["HMISystemDB".HMI_Axis.INPUT.Axis_ID].Par.SimplyTriggerPos := "HMISystemDB".HMI_Axis.INPUT.SimplyPos;
	    #IAI_Axis["HMISystemDB".HMI_Axis.INPUT.Axis_ID].Par.ListTrigger := "HMISystemDB".HMI_Axis.INPUT.ListTrigger;
	    #IAI_Axis["HMISystemDB".HMI_Axis.INPUT.Axis_ID].Par.ListPosID := "HMISystemDB".HMI_Axis.INPUT.ListPosID;
	    #IAI_Axis["HMISystemDB".HMI_Axis.INPUT.Axis_ID].Enable := "HMISystemDB".HMI_Axis.INPUT.Enable;
	    #IAI_Axis["HMISystemDB".HMI_Axis.INPUT.Axis_ID]."Jog+" := "HMISystemDB".HMI_Axis.INPUT."Jog+";
	    #IAI_Axis["HMISystemDB".HMI_Axis.INPUT.Axis_ID]."Jog-" := "HMISystemDB".HMI_Axis.INPUT."Jog-";
	    #IAI_Axis["HMISystemDB".HMI_Axis.INPUT.Axis_ID].Homing := "HMISystemDB".HMI_Axis.INPUT.Homing;
	    #IAI_Axis["HMISystemDB".HMI_Axis.INPUT.Axis_ID].Stop := "HMISystemDB".HMI_Axis.INPUT.Stop;
	END_IF;
	"HMISystemDB".HMI_Axis.OUTPUT.MAX_Axis := 3;
	"HMISystemDB".HMI_Axis.OUTPUT.Ready := #IAI_Axis["HMISystemDB".HMI_Axis.INPUT.Axis_ID].Ready;
	"HMISystemDB".HMI_Axis.OUTPUT.Alarm := #IAI_Axis["HMISystemDB".HMI_Axis.INPUT.Axis_ID].Error OR #IAI_Axis["HMISystemDB".HMI_Axis.INPUT.Axis_ID].OverTime;
	"HMISystemDB".HMI_Axis.OUTPUT.Warming := #IAI_Axis["HMISystemDB".HMI_Axis.INPUT.Axis_ID].Warn;
	"HMISystemDB".HMI_Axis.OUTPUT.RunEnd := #IAI_Axis["HMISystemDB".HMI_Axis.INPUT.Axis_ID].RunEnd;
	"HMISystemDB".HMI_Axis.OUTPUT.Interference := #IAI_Axis["HMISystemDB".HMI_Axis.INPUT.Axis_ID].InterfereEnable;
	"HMISystemDB".HMI_Axis.OUTPUT."Reference Point" := #IAI_Axis["HMISystemDB".HMI_Axis.INPUT.Axis_ID].Homed;
	"HMISystemDB".HMI_Axis.OUTPUT.CurrentPosition := #IAI_Axis["HMISystemDB".HMI_Axis.INPUT.Axis_ID].CurrentPosition;
	"HMISystemDB".HMI_Axis.OUTPUT.CurrentSpeed := #IAI_Axis["HMISystemDB".HMI_Axis.INPUT.Axis_ID].CurrentSpeed;
	"HMISystemDB".HMI_Axis.OUTPUT.Enable := #IAI_Axis["HMISystemDB".HMI_Axis.INPUT.Axis_ID].Enabled;
	"HMISystemDB".HMI_Axis.OUTPUT.TargetPosition := #IAI_Axis["HMISystemDB".HMI_Axis.INPUT.Axis_ID].Par.TargetPosition["HMISystemDB".HMI_Axis.INPUT.ListPosID];
	
	
	IF "ModeDB".Gen.Out.Change THEN
	    #IAI_Axis[1].Par.SimplyTriggerPos := 0.0;
	    #IAI_Axis[2].Par.SimplyTriggerPos := 0.0;
	    #IAI_Axis[3].Par.SimplyTriggerPos := 0.0;
	    "HMISystemDB".HMI_Axis.INPUT.SimplyPos := 0.0;
	END_IF;
	
	
	
	
	
	
	
	
END_FUNCTION_BLOCK

FUNCTION_BLOCK "IAI_BASE_FB"
{ S7_Optimized_Access := 'FALSE' }
VERSION : 0.1
   VAR_INPUT 
      Mode : "ModeGenStruct";
      "Input 4 word_Man1" : HW_IO;
      "Input 4 word_Man2" : HW_IO;
      "Input 4 word_1" : HW_IO;
      "Input 4 word_2" : HW_IO;
      "Output 4 word_Man1" : HW_IO;
      "Output 4 word_Man2" : HW_IO;
      "Output 4 word_1" : HW_IO;
      "Output 4 word_2" : HW_IO;
      Interfere : Bool;
      Axis_ID { ExternalAccessible := 'False'; ExternalVisible := 'False'; ExternalWritable := 'False'} : Int;
      AutoPointStart : Bool;
   END_VAR

   VAR_IN_OUT 
      Homing : Bool;
      AbsPos : Bool;
      RelaPos : Bool;
      Enable : Bool;
      Stop : Bool;
      "Jog+" : Bool;
      "Jog-" : Bool;
      PosCode : Int;
      RunEnd : Bool;
      Adjist : Bool;
   END_VAR

   VAR 
      Par { ExternalAccessible := 'False'; ExternalVisible := 'False'; ExternalWritable := 'False'} : Struct
         "Limit+" { ExternalAccessible := 'False'; ExternalVisible := 'False'; ExternalWritable := 'False'} : Bool;
         "Limit-" { ExternalAccessible := 'False'; ExternalVisible := 'False'; ExternalWritable := 'False'} : Bool;
         PositionWidth { ExternalAccessible := 'False'; ExternalVisible := 'False'; ExternalWritable := 'False'} : Real;
         PosCode { ExternalAccessible := 'False'; ExternalVisible := 'False'; ExternalWritable := 'False'} : Int;
         Speed { ExternalAccessible := 'False'; ExternalVisible := 'False'; ExternalWritable := 'False'} : Int;
         "Limt+Pos" { ExternalAccessible := 'False'; ExternalVisible := 'False'; ExternalWritable := 'False'} : Real;
         "Limt-Pos" { ExternalAccessible := 'False'; ExternalVisible := 'False'; ExternalWritable := 'False'} : Real;
         AccSpeed { ExternalAccessible := 'False'; ExternalVisible := 'False'; ExternalWritable := 'False'} : Int;
         DecSpeed { ExternalAccessible := 'False'; ExternalVisible := 'False'; ExternalWritable := 'False'} : Int;
         LuV { ExternalAccessible := 'False'; ExternalVisible := 'False'; ExternalWritable := 'False'} : Int;
         SimplyTrigger { ExternalAccessible := 'False'; ExternalVisible := 'False'; ExternalWritable := 'False'} : Bool;
         SimplyTriggerPos { ExternalAccessible := 'False'; ExternalVisible := 'False'; ExternalWritable := 'False'} : Real;
         ListTrigger { ExternalAccessible := 'False'; ExternalVisible := 'False'; ExternalWritable := 'False'} : Bool;
         ListPosID { ExternalAccessible := 'False'; ExternalVisible := 'False'; ExternalWritable := 'False'} : Int;
         TargetPosition { ExternalAccessible := 'False'; ExternalVisible := 'False'; ExternalWritable := 'False'} : Array[0..30] of Real;
         TargetSpeed { ExternalAccessible := 'False'; ExternalVisible := 'False'; ExternalWritable := 'False'} : Array[0..30] of Int;
         GoPosInterfere { ExternalAccessible := 'False'; ExternalVisible := 'False'; ExternalWritable := 'False'} : Array[0..30] of Bool;
         OverTime { ExternalAccessible := 'False'; ExternalVisible := 'False'; ExternalWritable := 'False'} : Time;
      END_STRUCT;
      RecvData : "IAI Input Struct";
      SendData : "IAI Output Struct";
      CurrentPosition : Real;
      CurrentSpeed : Int;
      TargetPosition : Real;
      Ready : Bool;
      Enabled : Bool;
      Homed : Bool;
      Error : Bool;
      Warn : Bool;
      HRunning : Bool;
      PRunning : Bool;
      Running : Bool;
      TemWritePos : Bool;
      TemGoPos : Bool;
      TemStart : Bool;
      RInterfere : Bool;
      PosInterfere : Bool;
      InterfereEnable : Bool;
      LimtStop : Bool;
      HomeJogTime {InstructionName := 'TON_TIME'; LibVersion := '1.0'} : TON_TIME;
      TemHomingok {InstructionName := 'TON_TIME'; LibVersion := '1.0'} : TON_TIME;
      TemPosOk {InstructionName := 'TON_TIME'; LibVersion := '1.0'} : TON_TIME;
      RunTime {InstructionName := 'TON_TIME'; LibVersion := '1.0'} : TON_TIME;
      RunSetTime : Time;
      OverTime : Bool;
      Cmd : Struct
         Homing : Bool;
         PosRun : Bool;
         Jog : Bool;
      END_STRUCT;
      Hstep : Int;
      Step : Int;
      PosTime {InstructionName := 'TON_TIME'; LibVersion := '1.0'} : TON_TIME;
      StopCmd : Bool;
      StopTime {InstructionName := 'TON_TIME'; LibVersion := '1.0'} : TON_TIME;
      Pos_ID : Int := 1;
      SetPosCode { S7_SetPoint := 'True'} : Int;
      AutoStart : Bool;
      TemPage { ExternalVisible := 'False'} : Int;
      TemGroup { ExternalVisible := 'False'} : Int;
      FOR_ID : Int;
      TemHMIClick : Bool;
      aRetvalRead { ExternalAccessible := 'False'; ExternalVisible := 'False'; ExternalWritable := 'False'} : Array[1..5] of Int;
      aRetvalWrite { ExternalAccessible := 'False'; ExternalVisible := 'False'; ExternalWritable := 'False'} : Array[1..5] of Int;
      PRunninDelay {InstructionName := 'TON_TIME'; LibVersion := '1.0'; S7_SetPoint := 'False'} : TON_TIME;
   END_VAR


BEGIN
	//=========================================================
	//========================输入映射=========================
	
	REGION 伺服赋值
	    // 获取网关状态
	    #aRetvalRead[1] := DPRD_DAT(LADDR := #"Input 4 word_Man1", RECORD => #RecvData."Input 4 word_Man1");
	    #aRetvalRead[2] := DPRD_DAT(LADDR := #"Input 4 word_Man2", RECORD => #RecvData."Input 4 word_Man2");
	    
	    // 获取轴状态
	    #aRetvalRead[3] := DPRD_DAT(LADDR := #"Input 4 word_1", RECORD => #RecvData."Input 4 word_1");
	    #aRetvalRead[4] := DPRD_DAT(LADDR := #"Input 4 word_2", RECORD => #RecvData."Input 4 word_2");
	    
	    #SendData."Output 4 word_2"."Accelerated Speed" := #Par.AccSpeed;  // 加速度    
	END_REGION
	REGION 电机功能检测及设定    
	    ////////////网关打开/////////////
	    #SendData."Output 4 word_Man1".Mon := TRUE;
	    //////////////伺服报警////////////////
	    IF #RecvData."Input 4 word_2".ALM OR #OverTime THEN
	        #Error := true;
	    END_IF;
	    //////////////软极限位检测停止/////////////
	    IF (#TargetPosition < #Par."Limt-Pos") OR (#TargetPosition > #Par."Limt+Pos") THEN
	        #LimtStop := true;
	    ELSE
	        #LimtStop := false;
	    END_IF;
	    ///////////触碰极限位置停止伺服运行///////
	    IF #LimtStop OR #Par."Limit+" OR #Par."Limit-" THEN
	        #Step := 0;
	        #Hstep := 0;
	        #AbsPos := false;
	        #RelaPos := false;
	    END_IF;
	    //////////////伺服报错终止运行///////////////
	    IF NOT #Mode.Out.Estop OR #RecvData."Input 4 word_2".ALM = TRUE THEN
	        #Hstep := 0;
	        #Step := 0;
	        #SendData."Output 4 word_2".STP := TRUE;
	        #Homing := false;
	        #TemStart := false;
	    END_IF;
	    ///////////////模式变化///////////////////
	    IF #Mode.Out.Change THEN
	        #SetPosCode := #Par.PosCode;
	        #Par.PosCode := #PosCode;
	        #"Jog-" := false;
	        #"Jog+" := false;
	        #Homing := false;
	        #AbsPos := false;
	        #RelaPos := false;
	        #Step := 0;
	        #Hstep := 0;
	    END_IF;
	    /////////位置代码干涉条件判断//////////////
	    IF #Par.ListTrigger OR #TemGoPos THEN
	        
	        IF #Par.GoPosInterfere[#Par.PosCode] THEN
	            #PosInterfere := true;
	        ELSE
	            #PosInterfere := false;
	        END_IF;
	    ELSE
	        #PosInterfere := true;
	    END_IF;
	    #RInterfere := #PosInterfere AND #Interfere;
	    ////////////干涉条件判断/////////////////////
	    IF #RInterfere OR #Adjist THEN
	        #InterfereEnable := true;
	    ELSE
	        #InterfereEnable := false;
	    END_IF;
	    //////////////轴使能//////////   
	    IF #Mode.Out.Estop AND #RecvData."Input 4 word_2".ALM = FALSE AND #Enable THEN //((#Mode.Out.Manual AND #Enable) OR #Mode.Out.Auto)
	        #SendData."Output 4 word_2".SON := TRUE;
	    ELSE
	        #SendData."Output 4 word_2".SON := FALSE;
	    END_IF;
	    ////////////使能反馈/////////////
	    IF #SendData."Output 4 word_2".SON AND #Mode.Out.Estop THEN
	        #Enabled := true;
	    ELSE
	        #Enabled := false;
	    END_IF;
	    ///////////轴报错初始化步骤/////////////
	    IF #Error THEN
	        #Step := 0;
	        #"Jog-" := false;
	        #"Jog+" := false;
	        #Hstep := 0;
	        #Homing := false;
	        #TemStart := false;
	    END_IF;
	    ////////////复位轴报警/////////
	    
	    IF #Mode.Out.Reset THEN
	        #Error := false;
	        #OverTime := FALSE;
	        #SendData."Output 4 word_2".RES := true;
	        #SendData."Output 4 word_2".Home := FALSE;
	        #Hstep := 0;
	        #SendData."Output 4 word_2".STP := FALSE;
	        //#SetPosCode := #Par.PosCode;
	    ELSE
	        #SendData."Output 4 word_2".RES := false;
	    END_IF;
	    //////////////Reday/////////////
	    IF #Enabled AND NOT #PRunning AND #Homed AND #InterfereEnable THEN
	        #Ready := true;
	    ELSE
	        #Ready := false;
	    END_IF;
	    /////////////////获取电机参数//////////////////////////
	    #"CurrentPosition" := DINT_TO_REAL(IN := #RecvData."Input 4 word_1"."Current Position") / 100;
	    #"CurrentSpeed" := #RecvData."Input 4 word_2"."Current Speed";
	    /////////////////电机速率设置/////////////
	    #SendData."Output 4 word_2".JVEL := TRUE;
	    #SendData."Output 4 word_1"."Location Width" := REAL_TO_DINT(IN := (#Par.PositionWidth * 100)); //宽度。
	END_REGION
	REGION 位置判断
	    IF #Mode.Out.Manual THEN
	        #FOR_ID := 0;
	    ELSE
	        #FOR_ID := 1;
	    END_IF;
	    
	    FOR #Pos_ID := #FOR_ID TO 29 DO
	        IF #CurrentPosition >= #Par.TargetPosition[#Pos_ID] - #Par.PositionWidth AND
	            #CurrentPosition <= #Par.TargetPosition[#Pos_ID] + #Par.PositionWidth AND #Homed THEN
	            #PosCode := #Pos_ID;
	            #SetPosCode := #Pos_ID;
	            EXIT;
	        ELSE
	            #PosCode := -9;
	        END_IF;
	    END_FOR;
	    
	END_REGION
	REGION 回原位
	    #TemHomingok(IN := #RecvData."Input 4 word_2".Hend AND #HRunning,    //原位ok时间
	                 PT := t#2s);
	    //////////////////执行程序////////////    
	    CASE #Hstep OF
	        0:
	            #HRunning := false;
	            IF #Homing AND #Enabled AND #InterfereEnable THEN
	                #SendData."Output 4 word_2".Home := TRUE;
	                #Step := 0;
	                #Homed := false;
	                #Hstep := 1;
	            END_IF;
	        1:  // Start Homing
	            IF (#RecvData."Input 4 word_2".Move = TRUE)
	            THEN
	                #HRunning := true;
	                #Hstep := 2;
	            END_IF;
	            
	        2:  // Home End
	            IF (#RecvData."Input 4 word_2".Hend = TRUE AND #TemHomingok.Q)
	            THEN
	                #SendData."Output 4 word_2".Home := FALSE;
	                #Hstep := 3;
	            END_IF;
	            
	        3:  // End of Chain
	            IF #SendData."Output 4 word_2".Home = FALSE THEN
	                #Homing := FALSE;
	                #Homed := TRUE;
	                #HRunning := FALSE;
	                #Hstep := 0;
	            END_IF;
	            
	    END_CASE;
	END_REGION
	REGION 定位控制 
	    /////////自动模式切换位置编号自动触发电机运行//////////  
	    //IF #Par.PosCode <> #SetPosCode THEN
	        IF (#Mode.Out.Auto OR #Mode.Out.Home) AND  #AutoPointStart THEN
	            #AutoStart := TRUE;
	        ELSE
	            #AutoStart := false;
	        END_IF;
	    //END_IF;
	    
	    IF #Mode.Out.Manual AND #Par.SimplyTrigger THEN
	        #Par.PosCode := 0;
	        #SetPosCode := #Par.PosCode;
	    ELSIF #Mode.Out.Manual AND #Par.ListTrigger THEN
	        #TargetPosition := #Par.TargetPosition[#Par.ListPosID];
	        #Par.PosCode := #Par.ListPosID;
	        #SetPosCode := #Par.PosCode;
	    END_IF;
	    
	    #Par.TargetPosition[0] := #Par.SimplyTriggerPos;
	    #Par.TargetSpeed[0] := #Par.Speed;
	    
	    IF #Mode.Out.Auto THEN
	        #TargetPosition := #Par.TargetPosition[#Par.PosCode];
	        #SendData."Output 4 word_1"."Target position" := REAL_TO_DINT(IN := (#TargetPosition * 100));//写入目标位置
	        #SendData."Output 4 word_2".Speed :=#Par.TargetSpeed[#Par.PosCode]; // 速度 
	    END_IF;
	    IF #Mode.Out.Manual THEN
	        
	        #SendData."Output 4 word_1"."Target position" := REAL_TO_DINT(IN := (#TargetPosition * 100));//写入目标位置
	        #SendData."Output 4 word_2".Speed := #Par.Speed;//#Par.TargetSpeed[#Par.ListPosID]; // 速度 
	    END_IF;
	(*    IF #Mode.Out.Manual AND #Par.PosCode = 0 THEN
	        #SendData."Output 4 word_2".Speed := #Par.TargetSpeed[0]; // 速度
	    ELSE
	        #SendData."Output 4 word_2".Speed := #Par.TargetSpeed[#Pos_ID]; // 速度 
	    END_IF; *)
	    //////////////////////触发启动/////////////
	    IF ((#Mode.Out.Manual AND (#Par.SimplyTrigger OR #Par.ListTrigger) AND #InterfereEnable AND #Par.Speed > 1.0))   // AND  #Par.PosCode = 0
	        OR ((#Mode.Out.Auto OR #Mode.Out.Home) AND #AutoStart AND #Mode.Out.Running AND #InterfereEnable AND #Par.Speed > 1.0) THEN
	        #TemStart := TRUE;
	    END_IF;
	    
	    CASE #Step OF
	        0:///////////////准备/////////////////// 
	            #PRunning := false;
	            #TemWritePos := false;
	            IF #TemStart AND #Ready AND #InterfereEnable THEN
	                #SendData."Output 4 word_2".STP := FALSE;
	                #RunEnd := false;
	                #"Jog-" := false;
	                #"Jog+" := false;
	                #Step := 1;
	            END_IF;
	        1://////////////目标位置//////////////////   
	            #PRunning := true;
	            IF #TemStart THEN       //定位位置
	                #TargetPosition := #Par.TargetPosition[#Par.PosCode];
	            END_IF;
	            IF #TargetPosition = #Par.TargetPosition[#Par.PosCode] THEN
	                #SendData."Output 4 word_1"."Target position" := REAL_TO_DINT(IN := (#TargetPosition * 100));//写入目标位置
	                #SendData."Output 4 word_2".Speed := #Par.TargetSpeed[#Par.PosCode]; // 速度 
	                IF #TargetPosition = #CurrentPosition THEN
	                    #PosCode := #Par.PosCode;
	                    #PRunning := FALSE;
	                    #TemStart := false;
	                    #RunEnd := TRUE;
	                    #SetPosCode := #Par.PosCode;
	                    IF #SetPosCode = #Par.PosCode THEN
	                        #Step := 0;
	                    END_IF;
	                ELSE
	                    #Step := 2;
	                END_IF;
	            END_IF;
	            
	        2: ///////////////启动///////////////////
	            #SendData."Output 4 word_1"."Target position" := REAL_TO_DINT(IN := (#TargetPosition * 100));//写入目标位置
	            #SendData."Output 4 word_2".Speed := #Par.TargetSpeed[#Par.PosCode]; // 速度 
	            IF #RecvData."Input 4 word_2".Pend AND "ClockMemory0.5s" AND #InterfereEnable THEN
	                #SendData."Output 4 word_2".CSTR := TRUE;
	            ELSE
	                #SendData."Output 4 word_2".CSTR := FALSE;
	            END_IF;
	            IF #RecvData."Input 4 word_2".Pend = FALSE AND #RecvData."Input 4 word_2".Move THEN //OR #TemPosOk.Q
	                #Step := 3;
	            END_IF;
	            
	        3: ///////////////////中间停止//////////////////
	            IF #Stop OR #InterfereEnable = FALSE THEN
	                #StopCmd := true;
	                #SendData."Output 4 word_2".STP := TRUE;
	            ELSE
	                #StopCmd := false;
	                #SendData."Output 4 word_2".STP := FALSE;
	            END_IF;
	            ////////////运行完成////////////////
	            IF #RecvData."Input 4 word_2".Pend THEN
	                #SendData."Output 4 word_2".CSTR := FALSE;
	                #Step := 4;
	            END_IF;
	        4: //////位置比较////////////
	            IF #Mode.Out.Manual THEN
	                
	                IF "IAI_DeviceCtl".IAIServo[#Axis_ID].Point[#Par.ListPosID].Achieve THEN
	                    #SetPosCode := #Par.PosCode;
	                    IF #SetPosCode = #Par.PosCode THEN
	                        ;
	                        #Step := 5;
	                    END_IF;
	                END_IF;
	                IF #RecvData."Input 4 word_1"."Current Position" = REAL_TO_DINT(IN := (#Par.SimplyTriggerPos * 100)) THEN
	                    #Step := 5;
	                END_IF;
	            END_IF;
	            IF #Mode.Out.Auto THEN
	                IF "IAI_DeviceCtl".IAIServo[#Axis_ID].Point[#Par.PosCode].Achieve THEN
	                    #SetPosCode := #Par.PosCode;
	                    IF #SetPosCode = #Par.PosCode THEN
	                        ;
	                        #Step := 5;
	                    END_IF;
	                END_IF;
	            END_IF;
	        5:
	            #SendData."Output 4 word_2".CSTR := FALSE;
	            #AutoStart := FALSE;
	            IF #SendData."Output 4 word_2".CSTR = FALSE AND #AutoStart = FALSE THEN
	                #RunEnd := true;
	                #PRunning := false;
	                #TemStart := FALSE;
	                #Step := 0;
	            END_IF;
	            
	    END_CASE;
	END_REGION
	///////////////////////////运行时间///////////////////////
	#Running := #HRunning OR #PRunning;
	#RunTime(IN := #Running,
	         PT := #RunSetTime);
	IF #RunTime.Q THEN
	    #OverTime := TRUE;
	END_IF;
	///////////////////JOG//////////////////
	REGION 点动控制
	    IF #Mode.Out.Manual AND #Step = 0 THEN
	        ;
	        
	        // #SendData.JISL := #"Jog+" OR #"Jog-";
	        /////////////////jog+////////////////
	        #SendData."Output 4 word_2"."JOG+" := #"Jog+" AND NOT #Par."Limit+" AND (#CurrentPosition < #Par."Limt+Pos");
	        /////////////////jog-///////////////
	        #SendData."Output 4 word_2"."JOG-" := #"Jog-" AND NOT #Par."Limit-" AND (#CurrentPosition > #Par."Limt-Pos");
	    END_IF;
	END_REGION
	
	//==========================================================
	//=========================输出映射=========================
	//==========================================================
	
	//网关控制
	#aRetvalWrite[1] := DPWR_DAT(LADDR := #"Output 4 word_Man1", RECORD := #SendData."Output 4 word_Man1");
	#aRetvalWrite[2] := DPWR_DAT(LADDR := #"Output 4 word_Man2", RECORD := #SendData."Output 4 word_Man2");
	
	//轴控制
	#aRetvalWrite[3] := DPWR_DAT(LADDR := #"Output 4 word_1", RECORD := #SendData."Output 4 word_1");
	#aRetvalWrite[4] := DPWR_DAT(LADDR := #"Output 4 word_2", RECORD := #SendData."Output 4 word_2");
	
	
	
	
	
	
	
	
END_FUNCTION_BLOCK

FUNCTION_BLOCK "KukaRobot1_Ctrl"
{ S7_Optimized_Access := 'FALSE' }
VERSION : 0.1
   VAR_INPUT 
      iHWID_In : HW_IO;
      iHWID_Out : HW_IO;
      iSysRun : Bool;
      iAuto : Bool;
      iManual : Bool;
      iSpecial : Bool;
      iE_STOP : Bool;
      iReset : Bool;
      iT1000ms : Bool;
      iTaskMode : USInt;
      iPartType : USInt;
      iSpeedValue : USInt;
      iPGNO : USInt;
   END_VAR

   VAR_OUTPUT 
      oReady : Bool;
      oStartComplete : Bool;
      oWarning : Bool;
      oError : Bool;
      oErrorCode : Int;
   END_VAR

   VAR_IN_OUT 
      ioAutoStart : Bool;
      ioSrartHome : Bool;
      ioStartAutoCycle : Bool;
   END_VAR

   VAR 
      sHMI : "KukaRobot_HMI";
      sROBtoPLC : Struct
         Sys : "KukaRobot_SysOutput";
         User : "KukaRobot_UserOutput_1";
      END_STRUCT;
      sPLCtoROB : Struct
         Sys : "KukaRobot_SysInput";
         User : "KukaRobot_UserInput_1";
      END_STRUCT;
      sDrivesOnDelay {InstructionName := 'TON_TIME'; LibVersion := '1.0'} : TON_TIME;
      sStartUpDelay {InstructionName := 'TON_TIME'; LibVersion := '1.0'} : TON_TIME;
      sRobotReadyToStart : Bool;
      sRobotReadyToRunning : Bool;
      sRobotActComplete : Bool;
      sRobotProgrameChoseOK : Bool;
      sSequence : Int;
      F_TRIG_Work {InstructionName := 'F_TRIG'; LibVersion := '1.0'} : F_TRIG;
      F_TRIG_Home {InstructionName := 'F_TRIG'; LibVersion := '1.0'} : F_TRIG;
      ModeValue : Int;
      Tem_ModeValue : Int;
      ModeChange : Bool;
      IEC_Timer_DRIVES_OFF {InstructionName := 'TON_TIME'; LibVersion := '1.0'} : TON_TIME;
      IEC_Timer_DRIVES_ON {InstructionName := 'TON_TIME'; LibVersion := '1.0'} : TON_TIME;
   END_VAR

   VAR_TEMP 
      tInRwENO : Bool;
      tOutRwENO : Bool;
      tInRwRetVal : Int;
      tOutRwRetVal : Int;
      "tROB-Input" : Array[1..128] of Byte;
      tROB_Output : Array[1..128] of Byte;
   END_VAR


BEGIN
	REGION Description
	    (*
	    %%%
	VERSION: V1.0
	LANGUAGE: ENGLISH
	    %%%
	    ** ** ** ** ** ** ** ** ** ** ** ** ** ** ** ** ** ** ** ** ** ** ** ** ** ** ** ** ** ** ** ** ** ** ** ** ** ** ** ** ** ** ** ** ** ** ** ** ** **
	    ** ** ** ** ** ** ** ** ** ** ** ** ** ** ** ** ** ** ** ** ** ** ** ** ** ** ** ** ** ** ** ** ** ** ** ** ** ** ** ** ** ** ** ** ** ** ** ** ** **
	    * *
	    * R (uhlamat) R (obot) I (nterface) *
	    * < < Robot Function Block > > *
	    * < < Handing Tool > > *
	    * - - - - - - - - - - - - - - - - - - - - - - - - - - - - - - - - - - - - - - - - - - *
	    * *
	    * Customer:   *
	    * Roboter Type: Kuka *
	    * Software: Siemens TIA V15.1 SP1 *
	    * Autor: ChenYi *
	    * Company: Ruhlamat Automation Technologies (Suzhou) Co., Ltd *
	    * Department: Elec.*
	    * Telephone: + 86 (512) 6767 1108 *
	    * *
	    * Version: 1.0 *
	    * Created: 26.05.2020 *
	    * Modified: 26.05.2020
	BY: ChenYi *
	    * *
	    ** ** ** ** ** ** ** ** ** ** ** ** ** ** ** ** ** ** ** ** ** ** ** ** ** ** ** ** ** ** ** ** ** ** ** ** ** ** ** ** ** ** ** ** ** ** ** ** ** **
	    ** ** ** ** ** ** ** ** ** ** ** ** ** ** ** ** ** ** ** ** ** ** ** ** ** ** ** ** ** ** ** ** ** ** ** ** ** ** ** ** ** ** ** ** ** ** ** ** ** **
	    %%%
	 #oErrorCode:
	    102:Robot home Failed
	    205:Failed to read HW Input data;
	    206:Failed to write HW Output data;
	    303:Start up TimeOut   
	    
	    %%%
	    *)
	END_REGION
	//<<<<<<<<<<<<<<<<<<<<<<<<<<<<<<<<<<<<<<<<<<<<<<<<<>>>>>>>>>>>>>>>>>>>>>>>>>>>>>>>>>>>>>>>>>>>>>>>>>
	//<<<<<<<<<<<<<<<<<<<<<<<<<<<<<<<<<<<<<<<<  Program Start  >>>>>>>>>>>>>>>>>>>>>>>>>>>>>>>>>>>>>>>>>
	//<<<<<<<<<<<<<<<<<<<<<<<<<<<<<<<<<<<<<<<<<<<<<<<<<>>>>>>>>>>>>>>>>>>>>>>>>>>>>>>>>>>>>>>>>>>>>>>>>>
	
	
	
	
	//******************************************
	REGION Bus Input Data Mapping
	    
	    #tInRwRetVal := DPRD_DAT(LADDR := #iHWID_In, RECORD => #sROBtoPLC, ENO => #tInRwENO);
	    IF NOT #tInRwENO THEN
	        GOTO ERROR;
	    END_IF;
	    
	END_REGION
	
	
	//******************************************
	(*Robot controller remmote control*)
	
	// I/O Act-Activate interface
	#sPLCtoROB.Sys.SI.I_O_ACT := 1;
	// Move Enable
	//#sPLCtoROB.Sys.SI.MOVE_ENABLE := (#iSysRun AND (((#sROBtoPLC.Sys.SO.T1 OR #sROBtoPLC.Sys.SO.T2) AND #iManual) OR (#iAuto))) AND #iSafePos;
	//#sPLCtoROB.Sys.SI.MOVE_ENABLE := #iSysRun AND (#iManual OR #iAuto) AND #iSafePos;
	IF #sROBtoPLC.Sys.SO.EXT = TRUE THEN
	    #sPLCtoROB.Sys.SI.MOVE_ENABLE := #iE_STOP;
	END_IF;
	IF #sROBtoPLC.Sys.SO.T1 = TRUE OR #sROBtoPLC.Sys.SO.T2 = TRUE THEN
	    #sPLCtoROB.Sys.SI.MOVE_ENABLE := TRUE;
	END_IF;
	// Drives Off
	#sPLCtoROB.Sys.SI.DRIVES_OFF := NOT #ModeChange;
	
	
	IF #iManual
	THEN
	    #ModeValue := 1;
	ELSIF #iAuto
	THEN
	    #ModeValue := 3;
	    
	END_IF;
	
	IF #ModeValue <> #Tem_ModeValue
	THEN
	    #ModeChange := true;
	ELSE
	    #ModeChange := false;
	END_IF;
	
	IF #IEC_Timer_DRIVES_OFF.Q THEN
	    #Tem_ModeValue := #ModeValue;
	END_IF;
	
	#IEC_Timer_DRIVES_OFF(IN:=#ModeValue <> #Tem_ModeValue,
	                      PT:=T#1s);
	
	
	//#sPLCtoROB.Sys.SI.DRIVES_OFF := #iSysRun;
	//#sPLCtoROB.Sys.SI.DRIVES_OFF := #iSysRun AND (#iManual OR #iAuto) AND #iSafePos;
	(*Robot controller ready to Start*)
	#sRobotReadyToStart := #iSysRun AND (#iAuto OR #iSpecial) AND
	#sROBtoPLC.Sys.SO.USER_SAF AND #sROBtoPLC.Sys.SO.ALARM_STOP AND
	#sROBtoPLC.Sys.SO.I_O_ACTCONF AND #sROBtoPLC.Sys.SO.ALARM_STOP_INTERN AND
	#sPLCtoROB.Sys.SI.MOVE_ENABLE AND #sPLCtoROB.Sys.SI.DRIVES_OFF
	AND #sROBtoPLC.Sys.SO.EXT;
	
	
	REGION Robot Start control
	    IF #sRobotReadyToStart THEN
	        IF (#sSequence = 0) AND #ioAutoStart AND (#iAuto OR #iSpecial) AND NOT #sRobotActComplete THEN
	            #sSequence := 100;
	            #ioAutoStart := 0;
	            #sRobotActComplete := 0;
	            #sRobotProgrameChoseOK := 0;
	        END_IF;
	        
	        #IEC_Timer_DRIVES_ON(IN := #sSequence=110,
	                              PT := T#100ms);
	        
	        CASE #sSequence OF
	(*            100:
	                #sPLCtoROB.Sys.SI.DRIVES_ON := 0;
	                #sSequence := 110;
	                
	            110:
	                #sPLCtoROB.Sys.SI.DRIVES_ON := 1;
	                IF #IEC_Timer_DRIVES_ON.Q THEN
	                    #sPLCtoROB.Sys.SI.DRIVES_ON := 0;
	                    #sSequence := 150;
	                END_IF;
	                *)
	            100:  // DrivesOn
	                IF NOT #sROBtoPLC.Sys.SO.RC_RDY1  THEN
	                        #sPLCtoROB.Sys.SI.CONF_MESS := 1;
	                        #sPLCtoROB.Sys.SI.DRIVES_ON := 0;
	                    ELSIF #sROBtoPLC.Sys.SO.RC_RDY1 THEN
	                        #sPLCtoROB.Sys.SI.CONF_MESS := 0;
	                        #sPLCtoROB.Sys.SI.DRIVES_ON := 1;
	                        IF #sDrivesOnDelay.Q AND #sROBtoPLC.Sys.SO.PERI_RDY THEN
	                            #sSequence := 200;
	                            #sPLCtoROB.Sys.SI.DRIVES_ON := 0;
	                            
	                        END_IF;
	                    END_IF;
	                    
	                    200:  // ALARM CONF
	                    IF #sROBtoPLC.Sys.SO.STOPMESS OR NOT #sROBtoPLC.Sys.SO.RC_RDY1 THEN
	                        #sPLCtoROB.Sys.SI.CONF_MESS := 1;
	                    ELSE
	                        #sPLCtoROB.Sys.SI.CONF_MESS := 0;
	                        #sSequence := 300;
	                    END_IF;
	                    
	                    300: // EXT_Start    
	                    IF #sROBtoPLC.Sys.SO.PERI_RDY AND NOT #sROBtoPLC.Sys.SO.STOPMESS THEN
	                        #sPLCtoROB.Sys.SI.EXT_START := 1;
	                        #sSequence := 400;
	                    END_IF;
	                    
	                    400: // EXT_Start Reset  
	                    IF #sROBtoPLC.Sys.SO.PRO_ACT THEN
	                        #sPLCtoROB.Sys.SI.EXT_START := 0;
	                        #sSequence := 500;
	                    END_IF;
	                    
	                    500: // Programe Call
	                    IF #sROBtoPLC.Sys.SO.PERI_RDY
	                        AND #sROBtoPLC.Sys.SO.PRO_ACT
	                        AND #sROBtoPLC.Sys.SO.PGNO_REQ
	                        AND #iPGNO <> 0
	                        //AND #s_ROBInput.User.User.Home.DI_AutoCycleStart
	                        //AND #s_ROBOutput.Sys."SO_$ON_PATH"
	                        //AND #s_ROBOutput.Sys."SO_$IN_HOME"
	                    THEN
	                        
	                        #sPLCtoROB.Sys.SI.PGNO_PBIT := #iPGNO;
	                        #sPLCtoROB.Sys.SI.PGNO_VALID := 1;
	                        #sSequence := 600;
	                    END_IF;
	                    
	                    600: // Programe Call Finish
	                    IF #sROBtoPLC.Sys.SO.APPL_RUN THEN
	                        #sPLCtoROB.Sys.SI.PGNO_VALID := 0;
	                        #sRobotActComplete := 1;
	                        #sSequence := 0;
	                    END_IF;
	                
	        END_CASE;
	        
	    ELSE
	        #sSequence := 0;
	        #sRobotActComplete := 0;
	//        #sPLCtoROB.Sys.SI.DRIVES_ON := 0;////2023/9/1更改
	        #sPLCtoROB.Sys.SI.EXT_START := 0;
	       // #sPLCtoROB.Sys.SI.CONF_MESS := 0;
	        #sPLCtoROB.Sys.SI.PGNO_VALID := 0;
	        #sPLCtoROB.Sys.SI.PGNO_PBIT := 0; 
	    END_IF;
	    
	(*Robot ready to Running*)
	    #sRobotReadyToRunning := #sRobotReadyToStart AND #sROBtoPLC.Sys.SO.PERI_RDY AND #sROBtoPLC.Sys.SO.PRO_ACT AND #sROBtoPLC.Sys.SO.APPL_RUN;
	    
	    
